REGION Network 42: Align Table Select Job
   // Decide which Step Sequence to start depending on the OMAC State and EM conditions
   // First Move Block is to Initialize the jobSelect Number
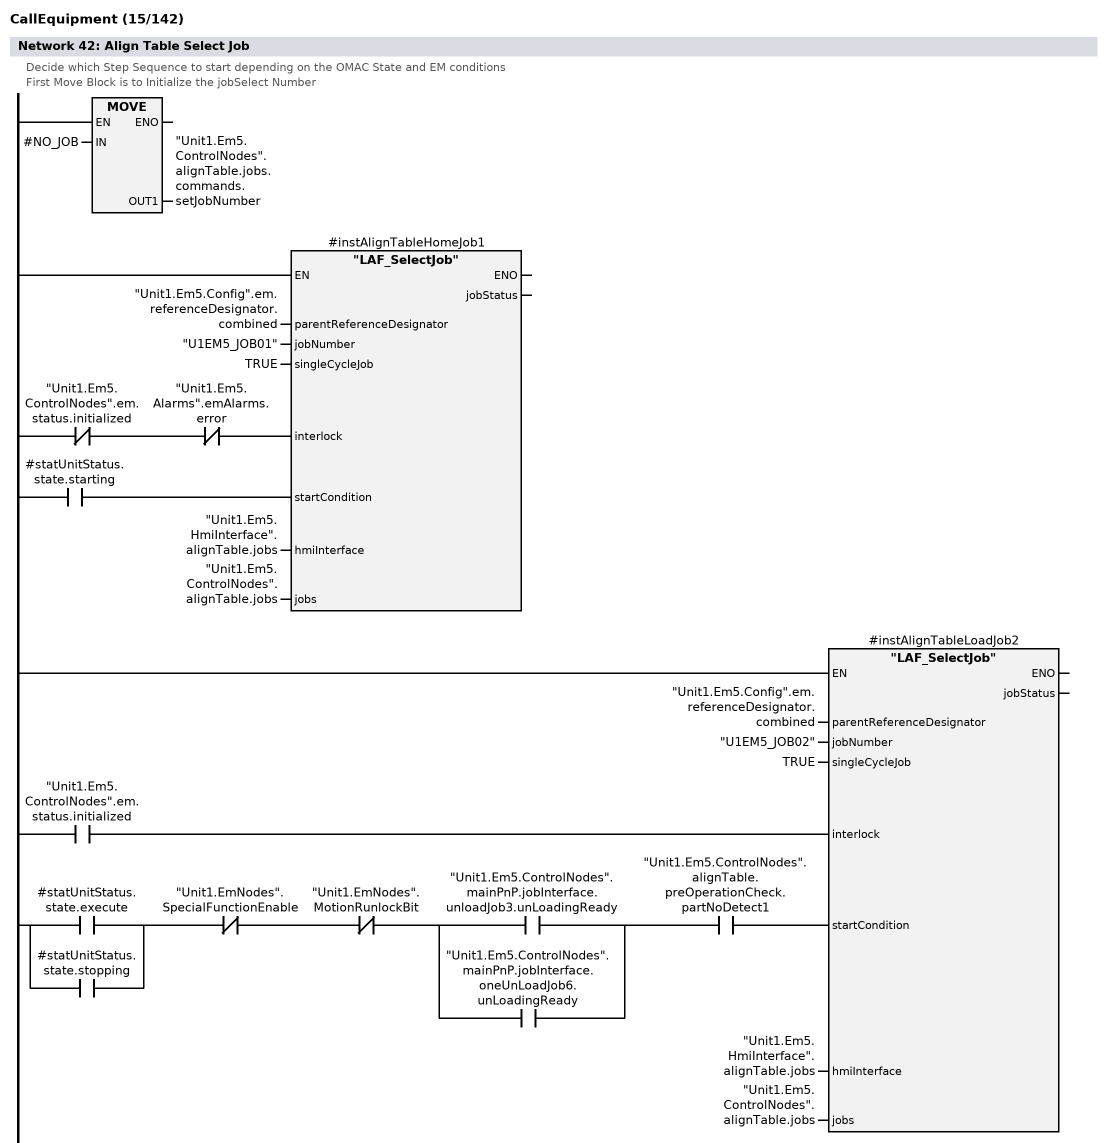
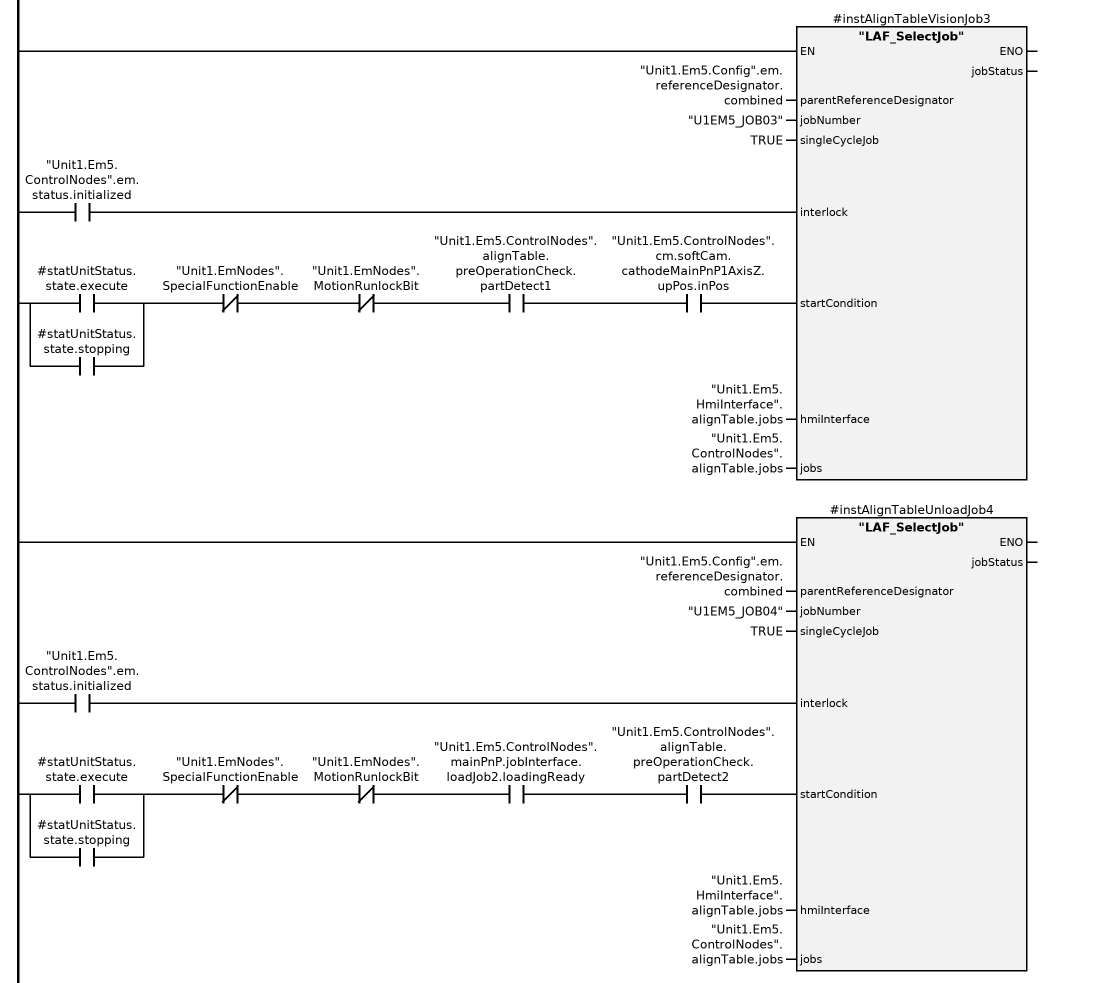
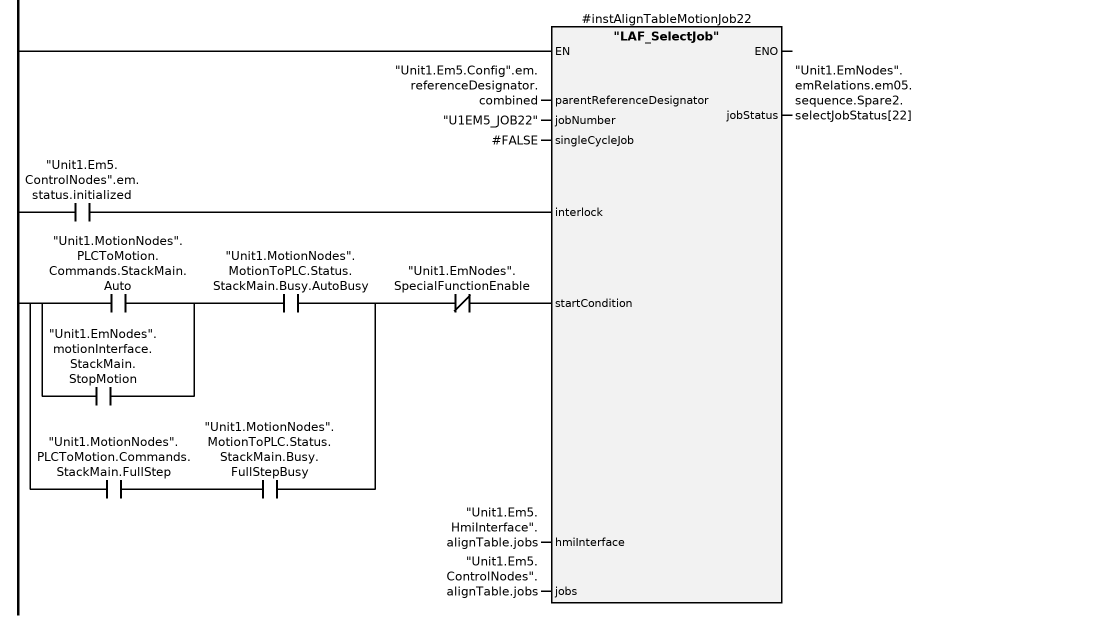
   RUNG wire#powerrail
      Move(in := #NO_JOB, out1 => "Unit1.Em5.ControlNodes".alignTable.jobs.commands.setJobNumber)
   END_RUNG
   RUNG wire#powerrail
      #instAlignTableHomeJob1(interlock := wire#w1, startCondition := wire#w2, parentReferenceDesignator := "Unit1.Em5.Config".em.referenceDesignator.combined, jobNumber := "U1EM5_JOB01", singleCycleJob := TRUE, hmiInterface := "Unit1.Em5.HmiInterface".alignTable.jobs, jobs := "Unit1.Em5.ControlNodes".alignTable.jobs, jobStatus =>)
   END_RUNG
   RUNG wire#powerrail
      I_Contact( "Unit1.Em5.ControlNodes".em.status.initialized )
      I_Contact( "Unit1.Em5.Alarms".emAlarms.error )
   END_RUNG wire#w1
   RUNG wire#powerrail
      Contact( #statUnitStatus.state.starting )
   END_RUNG wire#w2
   RUNG wire#powerrail
      #instAlignTableLoadJob2(interlock := wire#w3, startCondition := wire#w7, parentReferenceDesignator := "Unit1.Em5.Config".em.referenceDesignator.combined, jobNumber := "U1EM5_JOB02", singleCycleJob := TRUE, hmiInterface := "Unit1.Em5.HmiInterface".alignTable.jobs, jobs := "Unit1.Em5.ControlNodes".alignTable.jobs, jobStatus =>)
   END_RUNG
   RUNG wire#powerrail
      Contact( "Unit1.Em5.ControlNodes".em.status.initialized )
   END_RUNG wire#w3
   RUNG wire#powerrail
      Contact( #statUnitStatus.state.execute )
      wire#w4
      I_Contact( "Unit1.EmNodes".SpecialFunctionEnable )
      I_Contact( "Unit1.EmNodes".MotionRunlockBit )
      wire#w5
      Contact( "Unit1.Em5.ControlNodes".mainPnP.jobInterface.unloadJob3.unLoadingReady )
      wire#w6
      Contact( "Unit1.Em5.ControlNodes".alignTable.preOperationCheck.partNoDetect1 )
   END_RUNG wire#w7
   RUNG wire#powerrail
      Contact( #statUnitStatus.state.stopping )
   END_RUNG wire#w4
   RUNG wire#w5
      Contact( "Unit1.Em5.ControlNodes".mainPnP.jobInterface.oneUnLoadJob6.unLoadingReady )
   END_RUNG wire#w6
   RUNG wire#powerrail
      #instAlignTableVisionJob3(interlock := wire#w8, startCondition := wire#w10, parentReferenceDesignator := "Unit1.Em5.Config".em.referenceDesignator.combined, jobNumber := "U1EM5_JOB03", singleCycleJob := TRUE, hmiInterface := "Unit1.Em5.HmiInterface".alignTable.jobs, jobs := "Unit1.Em5.ControlNodes".alignTable.jobs, jobStatus =>)
   END_RUNG
   RUNG wire#powerrail
      Contact( "Unit1.Em5.ControlNodes".em.status.initialized )
   END_RUNG wire#w8
   RUNG wire#powerrail
      Contact( #statUnitStatus.state.execute )
      wire#w9
      I_Contact( "Unit1.EmNodes".SpecialFunctionEnable )
      I_Contact( "Unit1.EmNodes".MotionRunlockBit )
      Contact( "Unit1.Em5.ControlNodes".alignTable.preOperationCheck.partDetect1 )
      Contact( "Unit1.Em5.ControlNodes".cm.softCam.cathodeMainPnP1AxisZ.upPos.inPos )
   END_RUNG wire#w10
   RUNG wire#powerrail
      Contact( #statUnitStatus.state.stopping )
   END_RUNG wire#w9
   RUNG wire#powerrail
      #instAlignTableUnloadJob4(interlock := wire#w11, startCondition := wire#w13, parentReferenceDesignator := "Unit1.Em5.Config".em.referenceDesignator.combined, jobNumber := "U1EM5_JOB04", singleCycleJob := TRUE, hmiInterface := "Unit1.Em5.HmiInterface".alignTable.jobs, jobs := "Unit1.Em5.ControlNodes".alignTable.jobs, jobStatus =>)
   END_RUNG
   RUNG wire#powerrail
      Contact( "Unit1.Em5.ControlNodes".em.status.initialized )
   END_RUNG wire#w11
   RUNG wire#powerrail
      Contact( #statUnitStatus.state.execute )
      wire#w12
      I_Contact( "Unit1.EmNodes".SpecialFunctionEnable )
      I_Contact( "Unit1.EmNodes".MotionRunlockBit )
      Contact( "Unit1.Em5.ControlNodes".mainPnP.jobInterface.loadJob2.loadingReady )
      Contact( "Unit1.Em5.ControlNodes".alignTable.preOperationCheck.partDetect2 )
   END_RUNG wire#w13
   RUNG wire#powerrail
      Contact( #statUnitStatus.state.stopping )
   END_RUNG wire#w12
   RUNG wire#powerrail
      #instAlignTableMotionJob22(interlock := wire#w14, startCondition := wire#w17, parentReferenceDesignator := "Unit1.Em5.Config".em.referenceDesignator.combined, jobNumber := "U1EM5_JOB22", singleCycleJob := #FALSE, hmiInterface := "Unit1.Em5.HmiInterface".alignTable.jobs, jobs := "Unit1.Em5.ControlNodes".alignTable.jobs, jobStatus => "Unit1.EmNodes".emRelations.em05.sequence.Spare2.selectJobStatus[22])
   END_RUNG
   RUNG wire#powerrail
      Contact( "Unit1.Em5.ControlNodes".em.status.initialized )
   END_RUNG wire#w14
   RUNG wire#powerrail
      Contact( "Unit1.MotionNodes".PLCToMotion.Commands.StackMain.Auto )
      wire#w15
      Contact( "Unit1.MotionNodes".MotionToPLC.Status.StackMain.Busy.AutoBusy )
      wire#w16
      I_Contact( "Unit1.EmNodes".SpecialFunctionEnable )
   END_RUNG wire#w17
   RUNG wire#powerrail
      Contact( "Unit1.EmNodes".motionInterface.StackMain.StopMotion )
   END_RUNG wire#w15
   RUNG wire#powerrail
      Contact( "Unit1.MotionNodes".PLCToMotion.Commands.StackMain.FullStep )
      Contact( "Unit1.MotionNodes".MotionToPLC.Status.StackMain.Busy.FullStepBusy )
   END_RUNG wire#w16
   // the same network as SCL:
   "Unit1.Em5.ControlNodes".alignTable.jobs.commands.setJobNumber := #NO_JOB;
   #instAlignTableHomeJob1(parentReferenceDesignator := "Unit1.Em5.Config".em.referenceDesignator.combined,   // "LAF_SelectJob"
                           jobNumber := "U1EM5_JOB01",
                           singleCycleJob := TRUE,
                           interlock := NOT "Unit1.Em5.ControlNodes".em.status.initialized AND NOT "Unit1.Em5.Alarms".emAlarms.error,
                           startCondition := #statUnitStatus.state.starting,
                           hmiInterface := "Unit1.Em5.HmiInterface".alignTable.jobs,
                           jobs := "Unit1.Em5.ControlNodes".alignTable.jobs);
   #instAlignTableLoadJob2(parentReferenceDesignator := "Unit1.Em5.Config".em.referenceDesignator.combined,   // "LAF_SelectJob"
                           jobNumber := "U1EM5_JOB02",
                           singleCycleJob := TRUE,
                           interlock := "Unit1.Em5.ControlNodes".em.status.initialized,
                           startCondition := (#statUnitStatus.state.execute OR #statUnitStatus.state.stopping) AND NOT "Unit1.EmNodes".SpecialFunctionEnable AND NOT "Unit1.EmNodes".MotionRunlockBit AND ("Unit1.Em5.ControlNodes".mainPnP.jobInterface.unloadJob3.unLoadingReady OR "Unit1.Em5.ControlNodes".mainPnP.jobInterface.oneUnLoadJob6.unLoadingReady) AND "Unit1.Em5.ControlNodes".alignTable.preOperationCheck.partNoDetect1,
                           hmiInterface := "Unit1.Em5.HmiInterface".alignTable.jobs,
                           jobs := "Unit1.Em5.ControlNodes".alignTable.jobs);
   #instAlignTableVisionJob3(parentReferenceDesignator := "Unit1.Em5.Config".em.referenceDesignator.combined,   // "LAF_SelectJob"
                           jobNumber := "U1EM5_JOB03",
                           singleCycleJob := TRUE,
                           interlock := "Unit1.Em5.ControlNodes".em.status.initialized,
                           startCondition := (#statUnitStatus.state.execute OR #statUnitStatus.state.stopping) AND NOT "Unit1.EmNodes".SpecialFunctionEnable AND NOT "Unit1.EmNodes".MotionRunlockBit AND "Unit1.Em5.ControlNodes".alignTable.preOperationCheck.partDetect1 AND "Unit1.Em5.ControlNodes".cm.softCam.cathodeMainPnP1AxisZ.upPos.inPos,
                           hmiInterface := "Unit1.Em5.HmiInterface".alignTable.jobs,
                           jobs := "Unit1.Em5.ControlNodes".alignTable.jobs);
   #instAlignTableUnloadJob4(parentReferenceDesignator := "Unit1.Em5.Config".em.referenceDesignator.combined,   // "LAF_SelectJob"
                           jobNumber := "U1EM5_JOB04",
                           singleCycleJob := TRUE,
                           interlock := "Unit1.Em5.ControlNodes".em.status.initialized,
                           startCondition := (#statUnitStatus.state.execute OR #statUnitStatus.state.stopping) AND NOT "Unit1.EmNodes".SpecialFunctionEnable AND NOT "Unit1.EmNodes".MotionRunlockBit AND "Unit1.Em5.ControlNodes".mainPnP.jobInterface.loadJob2.loadingReady AND "Unit1.Em5.ControlNodes".alignTable.preOperationCheck.partDetect2,
                           hmiInterface := "Unit1.Em5.HmiInterface".alignTable.jobs,
                           jobs := "Unit1.Em5.ControlNodes".alignTable.jobs);
   #instAlignTableMotionJob22(parentReferenceDesignator := "Unit1.Em5.Config".em.referenceDesignator.combined,   // "LAF_SelectJob"
                           jobNumber := "U1EM5_JOB22",
                           singleCycleJob := #FALSE,
                           interlock := "Unit1.Em5.ControlNodes".em.status.initialized,
                           startCondition := ((("Unit1.MotionNodes".PLCToMotion.Commands.StackMain.Auto OR "Unit1.EmNodes".motionInterface.StackMain.StopMotion) AND "Unit1.MotionNodes".MotionToPLC.Status.StackMain.Busy.AutoBusy) OR ("Unit1.MotionNodes".PLCToMotion.Commands.StackMain.FullStep AND "Unit1.MotionNodes".MotionToPLC.Status.StackMain.Busy.FullStepBusy)) AND NOT "Unit1.EmNodes".SpecialFunctionEnable,
                           hmiInterface := "Unit1.Em5.HmiInterface".alignTable.jobs,
                           jobs := "Unit1.Em5.ControlNodes".alignTable.jobs,
                           jobStatus => "Unit1.EmNodes".emRelations.em05.sequence.Spare2.selectJobStatus[22]);
END_REGION

REGION Network 43: Align Table Job 1 Interface
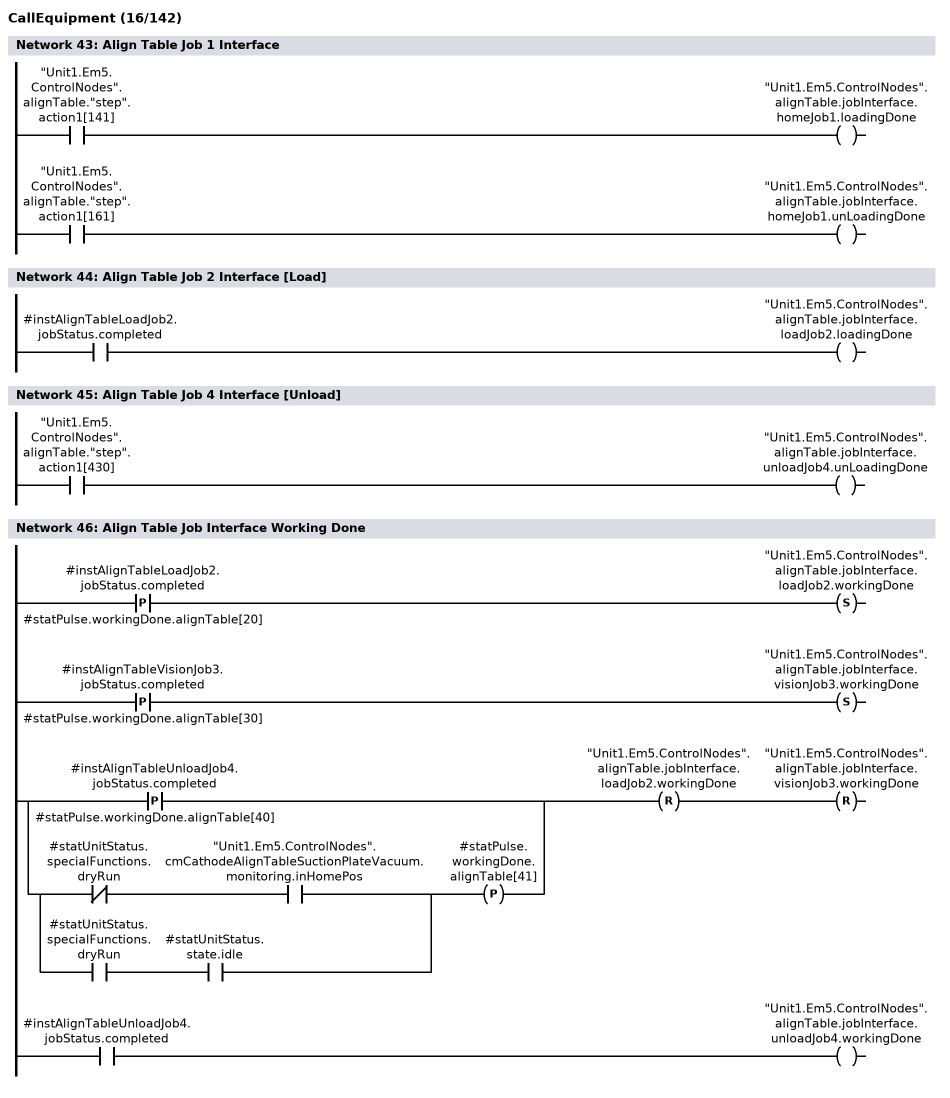
   RUNG wire#powerrail
      Contact( "Unit1.Em5.ControlNodes".alignTable."step".action1[141] )
      Coil( "Unit1.Em5.ControlNodes".alignTable.jobInterface.homeJob1.loadingDone )
   END_RUNG
   RUNG wire#powerrail
      Contact( "Unit1.Em5.ControlNodes".alignTable."step".action1[161] )
      Coil( "Unit1.Em5.ControlNodes".alignTable.jobInterface.homeJob1.unLoadingDone )
   END_RUNG
   // the same network as SCL:
   "Unit1.Em5.ControlNodes".alignTable.jobInterface.homeJob1.loadingDone := "Unit1.Em5.ControlNodes".alignTable."step".action1[141];
   "Unit1.Em5.ControlNodes".alignTable.jobInterface.homeJob1.unLoadingDone := "Unit1.Em5.ControlNodes".alignTable."step".action1[161];
END_REGION

REGION Network 44: Align Table Job 2 Interface [Load]
   RUNG wire#powerrail
      Contact( #instAlignTableLoadJob2.jobStatus.completed )
      Coil( "Unit1.Em5.ControlNodes".alignTable.jobInterface.loadJob2.loadingDone )
   END_RUNG
   // the same network as SCL:
   "Unit1.Em5.ControlNodes".alignTable.jobInterface.loadJob2.loadingDone := #instAlignTableLoadJob2.jobStatus.completed;
END_REGION

REGION Network 45: Align Table Job 4 Interface [Unload]
   RUNG wire#powerrail
      Contact( "Unit1.Em5.ControlNodes".alignTable."step".action1[430] )
      Coil( "Unit1.Em5.ControlNodes".alignTable.jobInterface.unloadJob4.unLoadingDone )
   END_RUNG
   // the same network as SCL:
   "Unit1.Em5.ControlNodes".alignTable.jobInterface.unloadJob4.unLoadingDone := "Unit1.Em5.ControlNodes".alignTable."step".action1[430];
END_REGION

REGION Network 46: Align Table Job Interface Working Done
   RUNG wire#powerrail
      P_Contact(operand := #instAlignTableLoadJob2.jobStatus.completed, bit := #statPulse.workingDone.alignTable[20])
      S_Coil( "Unit1.Em5.ControlNodes".alignTable.jobInterface.loadJob2.workingDone )
   END_RUNG
   RUNG wire#powerrail
      P_Contact(operand := #instAlignTableVisionJob3.jobStatus.completed, bit := #statPulse.workingDone.alignTable[30])
      S_Coil( "Unit1.Em5.ControlNodes".alignTable.jobInterface.visionJob3.workingDone )
   END_RUNG
   RUNG wire#powerrail
      P_Contact(operand := #instAlignTableUnloadJob4.jobStatus.completed, bit := #statPulse.workingDone.alignTable[40])
      wire#w1
      R_Coil( "Unit1.Em5.ControlNodes".alignTable.jobInterface.loadJob2.workingDone )
      R_Coil( "Unit1.Em5.ControlNodes".alignTable.jobInterface.visionJob3.workingDone )
   END_RUNG
   RUNG wire#powerrail
      I_Contact( #statUnitStatus.specialFunctions.dryRun )
      Contact( "Unit1.Em5.ControlNodes".cmCathodeAlignTableSuctionPlateVacuum.monitoring.inHomePos )
      wire#w2
      P_Trig( #statPulse.workingDone.alignTable[41] )
   END_RUNG wire#w1
   RUNG wire#powerrail
      Contact( #statUnitStatus.specialFunctions.dryRun )
      Contact( #statUnitStatus.state.idle )
   END_RUNG wire#w2
   RUNG wire#powerrail
      Contact( #instAlignTableUnloadJob4.jobStatus.completed )
      Coil( "Unit1.Em5.ControlNodes".alignTable.jobInterface.unloadJob4.workingDone )
   END_RUNG
   // the same network as SCL:
   #_w1 := #instAlignTableLoadJob2.jobStatus.completed AND NOT #statPulse.workingDone.alignTable[20];   // rising edge of #instAlignTableLoadJob2.jobStatus.completed
   #statPulse.workingDone.alignTable[20] := #instAlignTableLoadJob2.jobStatus.completed;
   IF #_w1 THEN "Unit1.Em5.ControlNodes".alignTable.jobInterface.loadJob2.workingDone := TRUE; END_IF;
   #_w2 := #instAlignTableVisionJob3.jobStatus.completed AND NOT #statPulse.workingDone.alignTable[30];   // rising edge of #instAlignTableVisionJob3.jobStatus.completed
   #statPulse.workingDone.alignTable[30] := #instAlignTableVisionJob3.jobStatus.completed;
   IF #_w2 THEN "Unit1.Em5.ControlNodes".alignTable.jobInterface.visionJob3.workingDone := TRUE; END_IF;
   #_w3 := #instAlignTableUnloadJob4.jobStatus.completed AND NOT #statPulse.workingDone.alignTable[40];   // rising edge of #instAlignTableUnloadJob4.jobStatus.completed
   #statPulse.workingDone.alignTable[40] := #instAlignTableUnloadJob4.jobStatus.completed;
   #_w4 := (NOT #statUnitStatus.specialFunctions.dryRun AND "Unit1.Em5.ControlNodes".cmCathodeAlignTableSuctionPlateVacuum.monitoring.inHomePos) OR (#statUnitStatus.specialFunctions.dryRun AND #statUnitStatus.state.idle);
   #_w5 := #_w4 AND NOT #statPulse.workingDone.alignTable[41];   // rising edge
   #statPulse.workingDone.alignTable[41] := #_w4;
   IF #_w3 OR #_w5 THEN
       "Unit1.Em5.ControlNodes".alignTable.jobInterface.loadJob2.workingDone := FALSE;
       "Unit1.Em5.ControlNodes".alignTable.jobInterface.visionJob3.workingDone := FALSE;
   END_IF;
   "Unit1.Em5.ControlNodes".alignTable.jobInterface.unloadJob4.workingDone := #instAlignTableUnloadJob4.jobStatus.completed;
END_REGION

REGION Network 47: Align Table Previous Operation Check
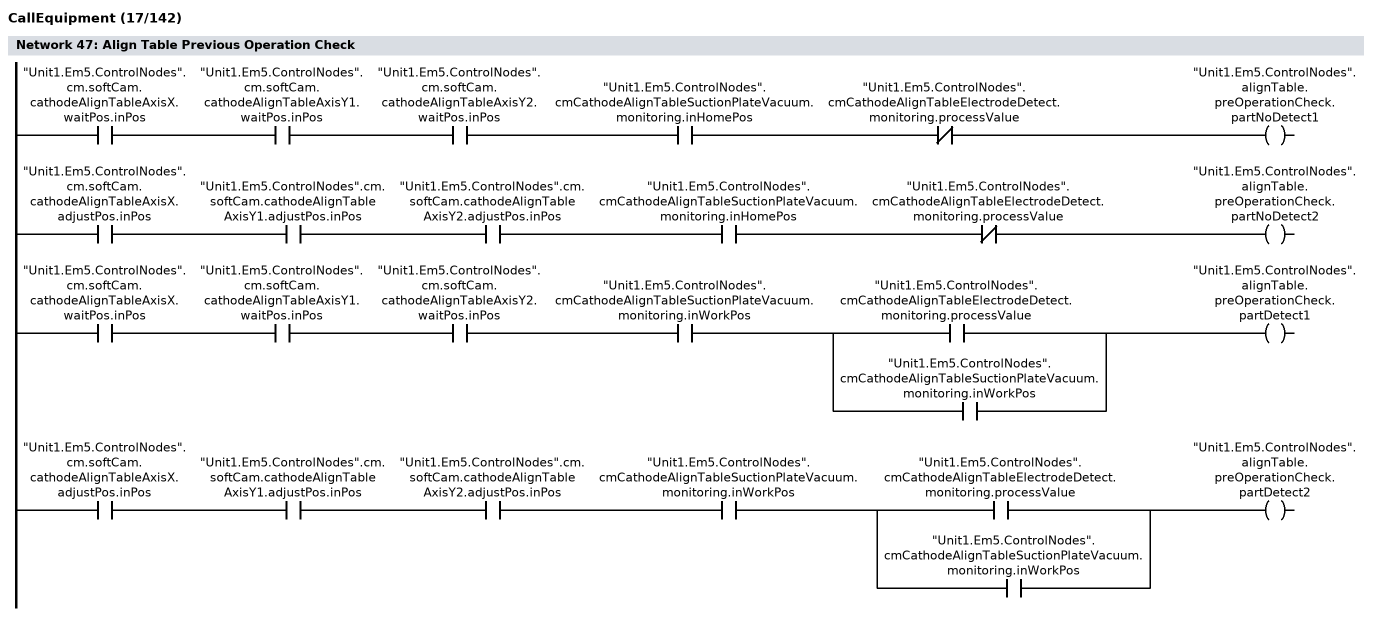
   RUNG wire#powerrail
      Contact( "Unit1.Em5.ControlNodes".cm.softCam.cathodeAlignTableAxisX.waitPos.inPos )
      Contact( "Unit1.Em5.ControlNodes".cm.softCam.cathodeAlignTableAxisY1.waitPos.inPos )
      Contact( "Unit1.Em5.ControlNodes".cm.softCam.cathodeAlignTableAxisY2.waitPos.inPos )
      Contact( "Unit1.Em5.ControlNodes".cmCathodeAlignTableSuctionPlateVacuum.monitoring.inHomePos )
      I_Contact( "Unit1.Em5.ControlNodes".cmCathodeAlignTableElectrodeDetect.monitoring.processValue )
      Coil( "Unit1.Em5.ControlNodes".alignTable.preOperationCheck.partNoDetect1 )
   END_RUNG
   RUNG wire#powerrail
      Contact( "Unit1.Em5.ControlNodes".cm.softCam.cathodeAlignTableAxisX.adjustPos.inPos )
      Contact( "Unit1.Em5.ControlNodes".cm.softCam.cathodeAlignTableAxisY1.adjustPos.inPos )
      Contact( "Unit1.Em5.ControlNodes".cm.softCam.cathodeAlignTableAxisY2.adjustPos.inPos )
      Contact( "Unit1.Em5.ControlNodes".cmCathodeAlignTableSuctionPlateVacuum.monitoring.inHomePos )
      I_Contact( "Unit1.Em5.ControlNodes".cmCathodeAlignTableElectrodeDetect.monitoring.processValue )
      Coil( "Unit1.Em5.ControlNodes".alignTable.preOperationCheck.partNoDetect2 )
   END_RUNG
   RUNG wire#powerrail
      Contact( "Unit1.Em5.ControlNodes".cm.softCam.cathodeAlignTableAxisX.waitPos.inPos )
      Contact( "Unit1.Em5.ControlNodes".cm.softCam.cathodeAlignTableAxisY1.waitPos.inPos )
      Contact( "Unit1.Em5.ControlNodes".cm.softCam.cathodeAlignTableAxisY2.waitPos.inPos )
      Contact( "Unit1.Em5.ControlNodes".cmCathodeAlignTableSuctionPlateVacuum.monitoring.inWorkPos )
      wire#w1
      Contact( "Unit1.Em5.ControlNodes".cmCathodeAlignTableElectrodeDetect.monitoring.processValue )
      wire#w2
      Coil( "Unit1.Em5.ControlNodes".alignTable.preOperationCheck.partDetect1 )
   END_RUNG
   RUNG wire#w1
      Contact( "Unit1.Em5.ControlNodes".cmCathodeAlignTableSuctionPlateVacuum.monitoring.inWorkPos )
   END_RUNG wire#w2
   RUNG wire#powerrail
      Contact( "Unit1.Em5.ControlNodes".cm.softCam.cathodeAlignTableAxisX.adjustPos.inPos )
      Contact( "Unit1.Em5.ControlNodes".cm.softCam.cathodeAlignTableAxisY1.adjustPos.inPos )
      Contact( "Unit1.Em5.ControlNodes".cm.softCam.cathodeAlignTableAxisY2.adjustPos.inPos )
      Contact( "Unit1.Em5.ControlNodes".cmCathodeAlignTableSuctionPlateVacuum.monitoring.inWorkPos )
      wire#w3
      Contact( "Unit1.Em5.ControlNodes".cmCathodeAlignTableElectrodeDetect.monitoring.processValue )
      wire#w4
      Coil( "Unit1.Em5.ControlNodes".alignTable.preOperationCheck.partDetect2 )
   END_RUNG
   RUNG wire#w3
      Contact( "Unit1.Em5.ControlNodes".cmCathodeAlignTableSuctionPlateVacuum.monitoring.inWorkPos )
   END_RUNG wire#w4
   // the same network as SCL:
   "Unit1.Em5.ControlNodes".alignTable.preOperationCheck.partNoDetect1 := "Unit1.Em5.ControlNodes".cm.softCam.cathodeAlignTableAxisX.waitPos.inPos AND "Unit1.Em5.ControlNodes".cm.softCam.cathodeAlignTableAxisY1.waitPos.inPos AND "Unit1.Em5.ControlNodes".cm.softCam.cathodeAlignTableAxisY2.waitPos.inPos AND "Unit1.Em5.ControlNodes".cmCathodeAlignTableSuctionPlateVacuum.monitoring.inHomePos AND NOT "Unit1.Em5.ControlNodes".cmCathodeAlignTableElectrodeDetect.monitoring.processValue;
   "Unit1.Em5.ControlNodes".alignTable.preOperationCheck.partNoDetect2 := "Unit1.Em5.ControlNodes".cm.softCam.cathodeAlignTableAxisX.adjustPos.inPos AND "Unit1.Em5.ControlNodes".cm.softCam.cathodeAlignTableAxisY1.adjustPos.inPos AND "Unit1.Em5.ControlNodes".cm.softCam.cathodeAlignTableAxisY2.adjustPos.inPos AND "Unit1.Em5.ControlNodes".cmCathodeAlignTableSuctionPlateVacuum.monitoring.inHomePos AND NOT "Unit1.Em5.ControlNodes".cmCathodeAlignTableElectrodeDetect.monitoring.processValue;
   "Unit1.Em5.ControlNodes".alignTable.preOperationCheck.partDetect1 := "Unit1.Em5.ControlNodes".cm.softCam.cathodeAlignTableAxisX.waitPos.inPos AND "Unit1.Em5.ControlNodes".cm.softCam.cathodeAlignTableAxisY1.waitPos.inPos AND "Unit1.Em5.ControlNodes".cm.softCam.cathodeAlignTableAxisY2.waitPos.inPos AND "Unit1.Em5.ControlNodes".cmCathodeAlignTableSuctionPlateVacuum.monitoring.inWorkPos AND ("Unit1.Em5.ControlNodes".cmCathodeAlignTableElectrodeDetect.monitoring.processValue OR "Unit1.Em5.ControlNodes".cmCathodeAlignTableSuctionPlateVacuum.monitoring.inWorkPos);
   "Unit1.Em5.ControlNodes".alignTable.preOperationCheck.partDetect2 := "Unit1.Em5.ControlNodes".cm.softCam.cathodeAlignTableAxisX.adjustPos.inPos AND "Unit1.Em5.ControlNodes".cm.softCam.cathodeAlignTableAxisY1.adjustPos.inPos AND "Unit1.Em5.ControlNodes".cm.softCam.cathodeAlignTableAxisY2.adjustPos.inPos AND "Unit1.Em5.ControlNodes".cmCathodeAlignTableSuctionPlateVacuum.monitoring.inWorkPos AND ("Unit1.Em5.ControlNodes".cmCathodeAlignTableElectrodeDetect.monitoring.processValue OR "Unit1.Em5.ControlNodes".cmCathodeAlignTableSuctionPlateVacuum.monitoring.inWorkPos);
END_REGION

REGION Network 49: NG P&P Select Job
   // Decide which Step Sequence to start depending on the OMAC State and EM conditions
   // First Move Block is to Initialize the jobSelect Number
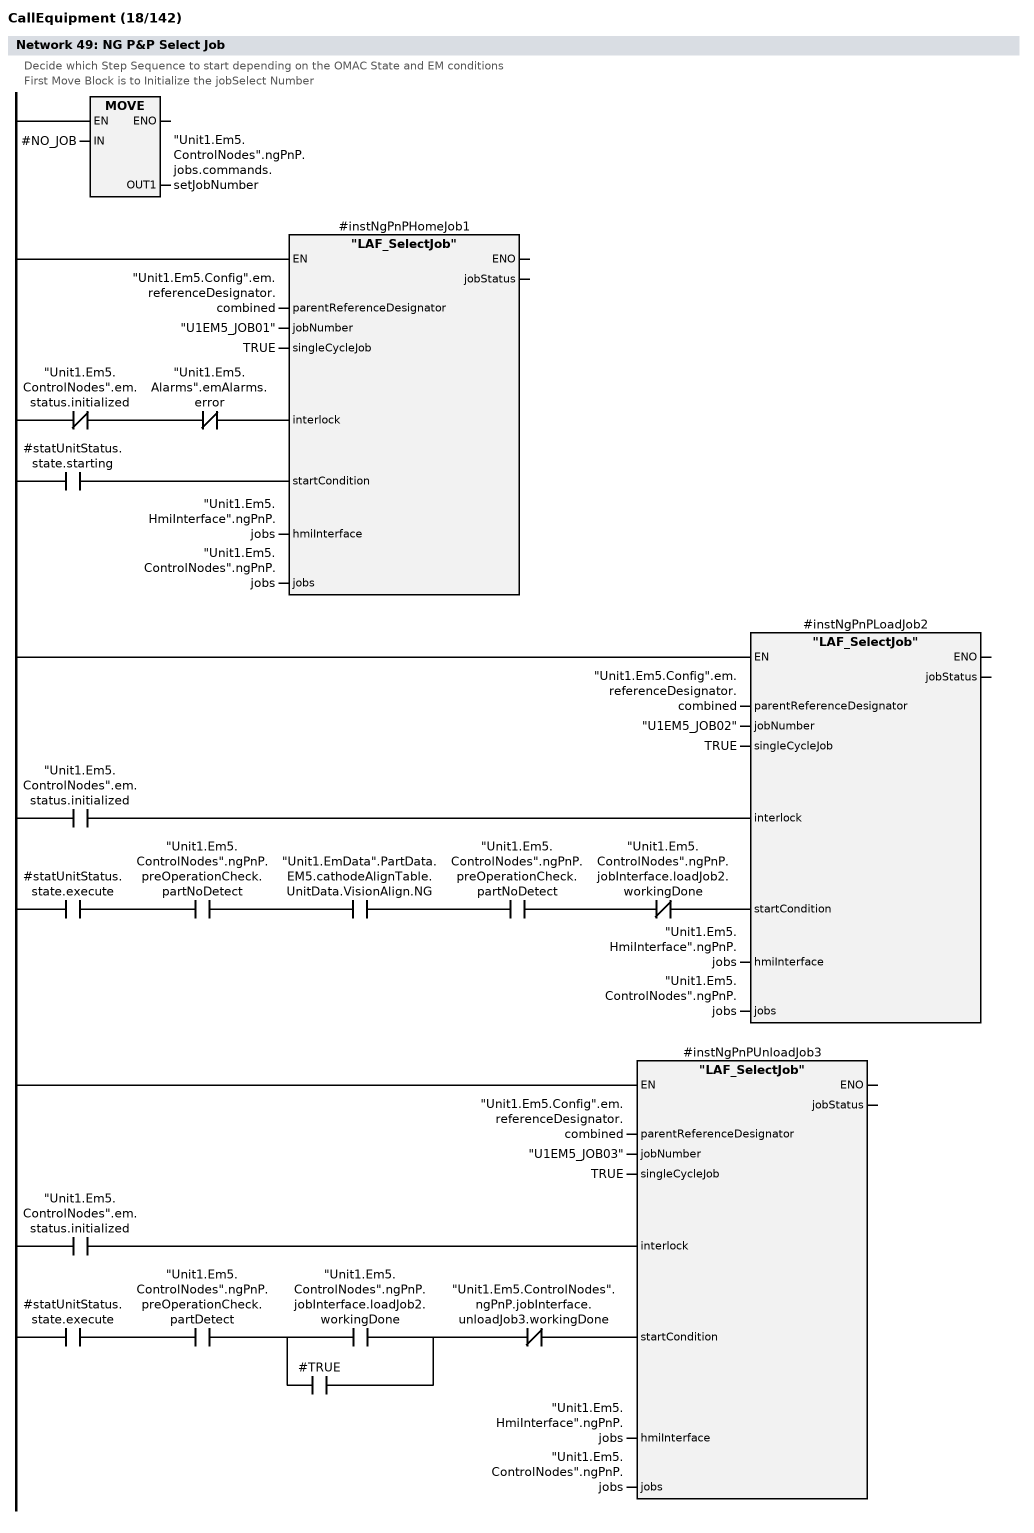
   RUNG wire#powerrail
      Move(in := #NO_JOB, out1 => "Unit1.Em5.ControlNodes".ngPnP.jobs.commands.setJobNumber)
   END_RUNG
   RUNG wire#powerrail
      #instNgPnPHomeJob1(interlock := wire#w1, startCondition := wire#w2, parentReferenceDesignator := "Unit1.Em5.Config".em.referenceDesignator.combined, jobNumber := "U1EM5_JOB01", singleCycleJob := TRUE, hmiInterface := "Unit1.Em5.HmiInterface".ngPnP.jobs, jobs := "Unit1.Em5.ControlNodes".ngPnP.jobs, jobStatus =>)
   END_RUNG
   RUNG wire#powerrail
      I_Contact( "Unit1.Em5.ControlNodes".em.status.initialized )
      I_Contact( "Unit1.Em5.Alarms".emAlarms.error )
   END_RUNG wire#w1
   RUNG wire#powerrail
      Contact( #statUnitStatus.state.starting )
   END_RUNG wire#w2
   RUNG wire#powerrail
      #instNgPnPLoadJob2(interlock := wire#w3, startCondition := wire#w4, parentReferenceDesignator := "Unit1.Em5.Config".em.referenceDesignator.combined, jobNumber := "U1EM5_JOB02", singleCycleJob := TRUE, hmiInterface := "Unit1.Em5.HmiInterface".ngPnP.jobs, jobs := "Unit1.Em5.ControlNodes".ngPnP.jobs, jobStatus =>)
   END_RUNG
   RUNG wire#powerrail
      Contact( "Unit1.Em5.ControlNodes".em.status.initialized )
   END_RUNG wire#w3
   RUNG wire#powerrail
      Contact( #statUnitStatus.state.execute )
      Contact( "Unit1.Em5.ControlNodes".ngPnP.preOperationCheck.partNoDetect )
      Contact( "Unit1.EmData".PartData.EM5.cathodeAlignTable.UnitData.VisionAlign.NG )
      Contact( "Unit1.Em5.ControlNodes".ngPnP.preOperationCheck.partNoDetect )
      I_Contact( "Unit1.Em5.ControlNodes".ngPnP.jobInterface.loadJob2.workingDone )
   END_RUNG wire#w4
   RUNG wire#powerrail
      #instNgPnPUnloadJob3(interlock := wire#w5, startCondition := wire#w8, parentReferenceDesignator := "Unit1.Em5.Config".em.referenceDesignator.combined, jobNumber := "U1EM5_JOB03", singleCycleJob := TRUE, hmiInterface := "Unit1.Em5.HmiInterface".ngPnP.jobs, jobs := "Unit1.Em5.ControlNodes".ngPnP.jobs, jobStatus =>)
   END_RUNG
   RUNG wire#powerrail
      Contact( "Unit1.Em5.ControlNodes".em.status.initialized )
   END_RUNG wire#w5
   RUNG wire#powerrail
      Contact( #statUnitStatus.state.execute )
      Contact( "Unit1.Em5.ControlNodes".ngPnP.preOperationCheck.partDetect )
      wire#w6
      Contact( "Unit1.Em5.ControlNodes".ngPnP.jobInterface.loadJob2.workingDone )
      wire#w7
      I_Contact( "Unit1.Em5.ControlNodes".ngPnP.jobInterface.unloadJob3.workingDone )
   END_RUNG wire#w8
   RUNG wire#w6
      Contact( #TRUE )
   END_RUNG wire#w7
   // the same network as SCL:
   "Unit1.Em5.ControlNodes".ngPnP.jobs.commands.setJobNumber := #NO_JOB;
   #instNgPnPHomeJob1(parentReferenceDesignator := "Unit1.Em5.Config".em.referenceDesignator.combined,   // "LAF_SelectJob"
                      jobNumber := "U1EM5_JOB01",
                      singleCycleJob := TRUE,
                      interlock := NOT "Unit1.Em5.ControlNodes".em.status.initialized AND NOT "Unit1.Em5.Alarms".emAlarms.error,
                      startCondition := #statUnitStatus.state.starting,
                      hmiInterface := "Unit1.Em5.HmiInterface".ngPnP.jobs,
                      jobs := "Unit1.Em5.ControlNodes".ngPnP.jobs);
   #instNgPnPLoadJob2(parentReferenceDesignator := "Unit1.Em5.Config".em.referenceDesignator.combined,   // "LAF_SelectJob"
                      jobNumber := "U1EM5_JOB02",
                      singleCycleJob := TRUE,
                      interlock := "Unit1.Em5.ControlNodes".em.status.initialized,
                      startCondition := #statUnitStatus.state.execute AND "Unit1.Em5.ControlNodes".ngPnP.preOperationCheck.partNoDetect AND "Unit1.EmData".PartData.EM5.cathodeAlignTable.UnitData.VisionAlign.NG AND "Unit1.Em5.ControlNodes".ngPnP.preOperationCheck.partNoDetect AND NOT "Unit1.Em5.ControlNodes".ngPnP.jobInterface.loadJob2.workingDone,
                      hmiInterface := "Unit1.Em5.HmiInterface".ngPnP.jobs,
                      jobs := "Unit1.Em5.ControlNodes".ngPnP.jobs);
   #instNgPnPUnloadJob3(parentReferenceDesignator := "Unit1.Em5.Config".em.referenceDesignator.combined,   // "LAF_SelectJob"
                        jobNumber := "U1EM5_JOB03",
                        singleCycleJob := TRUE,
                        interlock := "Unit1.Em5.ControlNodes".em.status.initialized,
                        startCondition := #statUnitStatus.state.execute AND "Unit1.Em5.ControlNodes".ngPnP.preOperationCheck.partDetect AND ("Unit1.Em5.ControlNodes".ngPnP.jobInterface.loadJob2.workingDone OR #TRUE) AND NOT "Unit1.Em5.ControlNodes".ngPnP.jobInterface.unloadJob3.workingDone,
                        hmiInterface := "Unit1.Em5.HmiInterface".ngPnP.jobs,
                        jobs := "Unit1.Em5.ControlNodes".ngPnP.jobs);
END_REGION

REGION Network 50: NG P&P Job 1 Interface
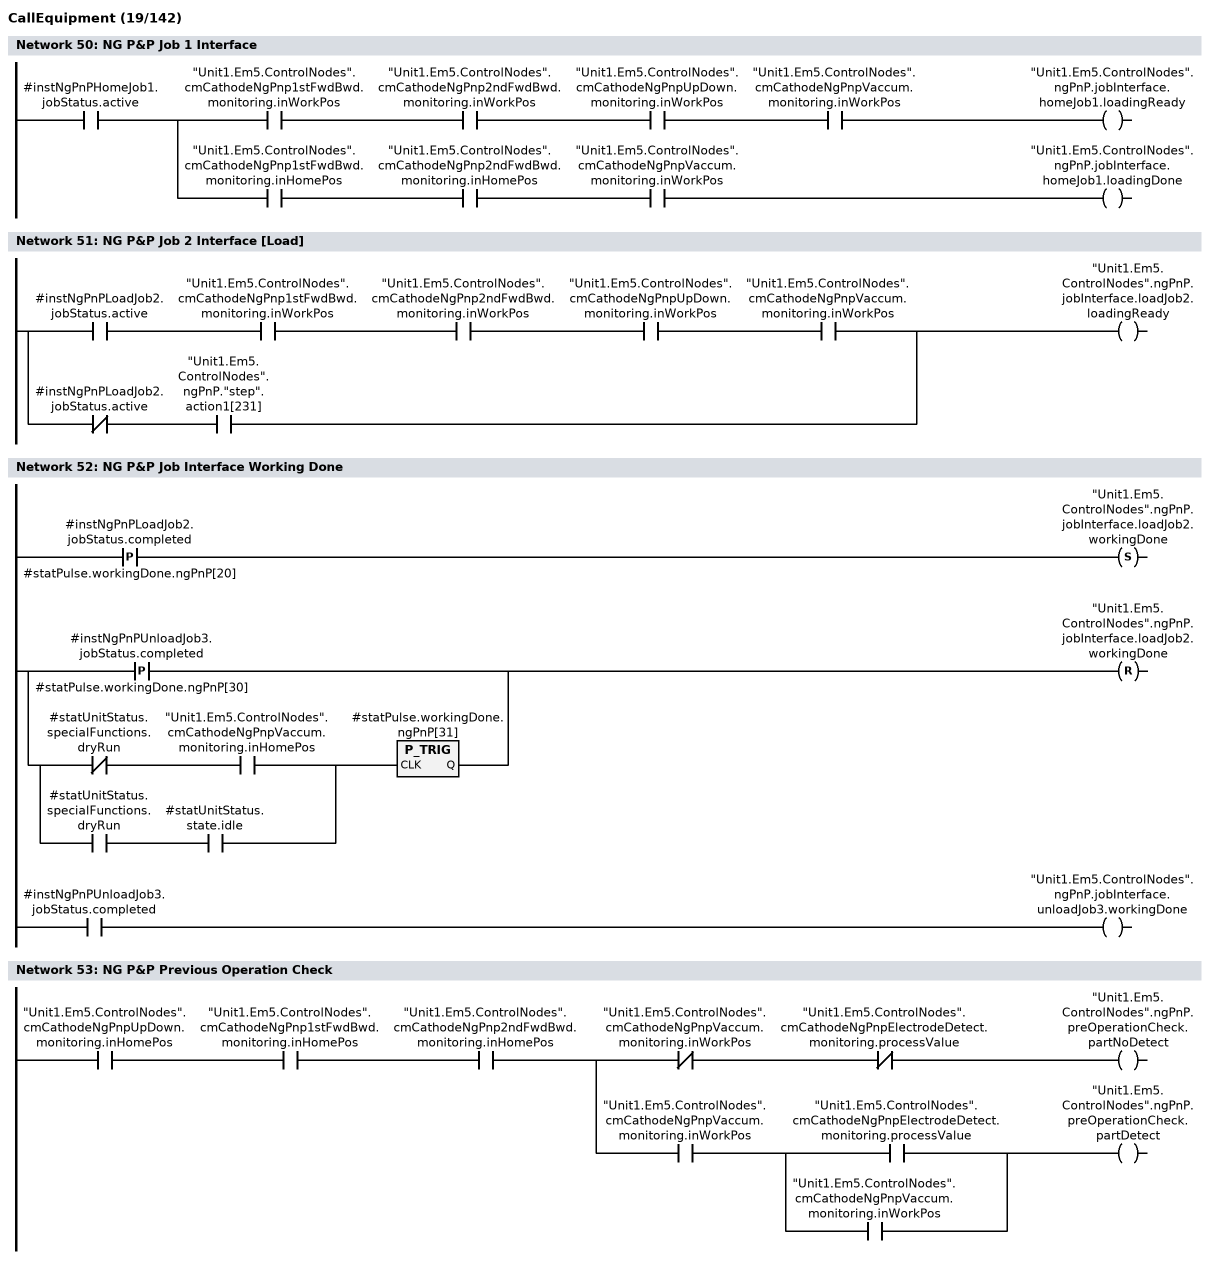
   RUNG wire#powerrail
      Contact( #instNgPnPHomeJob1.jobStatus.active )
      wire#w1
      Contact( "Unit1.Em5.ControlNodes".cmCathodeNgPnp1stFwdBwd.monitoring.inWorkPos )
      Contact( "Unit1.Em5.ControlNodes".cmCathodeNgPnp2ndFwdBwd.monitoring.inWorkPos )
      Contact( "Unit1.Em5.ControlNodes".cmCathodeNgPnpUpDown.monitoring.inWorkPos )
      Contact( "Unit1.Em5.ControlNodes".cmCathodeNgPnpVaccum.monitoring.inWorkPos )
      Coil( "Unit1.Em5.ControlNodes".ngPnP.jobInterface.homeJob1.loadingReady )
   END_RUNG
   RUNG wire#w1
      Contact( "Unit1.Em5.ControlNodes".cmCathodeNgPnp1stFwdBwd.monitoring.inHomePos )
      Contact( "Unit1.Em5.ControlNodes".cmCathodeNgPnp2ndFwdBwd.monitoring.inHomePos )
      Contact( "Unit1.Em5.ControlNodes".cmCathodeNgPnpVaccum.monitoring.inWorkPos )
      Coil( "Unit1.Em5.ControlNodes".ngPnP.jobInterface.homeJob1.loadingDone )
   END_RUNG
   // the same network as SCL:
   "Unit1.Em5.ControlNodes".ngPnP.jobInterface.homeJob1.loadingReady := #instNgPnPHomeJob1.jobStatus.active AND "Unit1.Em5.ControlNodes".cmCathodeNgPnp1stFwdBwd.monitoring.inWorkPos AND "Unit1.Em5.ControlNodes".cmCathodeNgPnp2ndFwdBwd.monitoring.inWorkPos AND "Unit1.Em5.ControlNodes".cmCathodeNgPnpUpDown.monitoring.inWorkPos AND "Unit1.Em5.ControlNodes".cmCathodeNgPnpVaccum.monitoring.inWorkPos;
   "Unit1.Em5.ControlNodes".ngPnP.jobInterface.homeJob1.loadingDone := #instNgPnPHomeJob1.jobStatus.active AND "Unit1.Em5.ControlNodes".cmCathodeNgPnp1stFwdBwd.monitoring.inHomePos AND "Unit1.Em5.ControlNodes".cmCathodeNgPnp2ndFwdBwd.monitoring.inHomePos AND "Unit1.Em5.ControlNodes".cmCathodeNgPnpVaccum.monitoring.inWorkPos;
END_REGION

REGION Network 51: NG P&P Job 2 Interface [Load]
   RUNG wire#powerrail
      Contact( #instNgPnPLoadJob2.jobStatus.active )
      Contact( "Unit1.Em5.ControlNodes".cmCathodeNgPnp1stFwdBwd.monitoring.inWorkPos )
      Contact( "Unit1.Em5.ControlNodes".cmCathodeNgPnp2ndFwdBwd.monitoring.inWorkPos )
      Contact( "Unit1.Em5.ControlNodes".cmCathodeNgPnpUpDown.monitoring.inWorkPos )
      Contact( "Unit1.Em5.ControlNodes".cmCathodeNgPnpVaccum.monitoring.inWorkPos )
      wire#w1
      Coil( "Unit1.Em5.ControlNodes".ngPnP.jobInterface.loadJob2.loadingReady )
   END_RUNG
   RUNG wire#powerrail
      I_Contact( #instNgPnPLoadJob2.jobStatus.active )
      Contact( "Unit1.Em5.ControlNodes".ngPnP."step".action1[231] )
   END_RUNG wire#w1
   // the same network as SCL:
   "Unit1.Em5.ControlNodes".ngPnP.jobInterface.loadJob2.loadingReady := (#instNgPnPLoadJob2.jobStatus.active AND "Unit1.Em5.ControlNodes".cmCathodeNgPnp1stFwdBwd.monitoring.inWorkPos AND "Unit1.Em5.ControlNodes".cmCathodeNgPnp2ndFwdBwd.monitoring.inWorkPos AND "Unit1.Em5.ControlNodes".cmCathodeNgPnpUpDown.monitoring.inWorkPos AND "Unit1.Em5.ControlNodes".cmCathodeNgPnpVaccum.monitoring.inWorkPos) OR (NOT #instNgPnPLoadJob2.jobStatus.active AND "Unit1.Em5.ControlNodes".ngPnP."step".action1[231]);
END_REGION

REGION Network 52: NG P&P Job Interface Working Done
   RUNG wire#powerrail
      P_Contact(operand := #instNgPnPLoadJob2.jobStatus.completed, bit := #statPulse.workingDone.ngPnP[20])
      S_Coil( "Unit1.Em5.ControlNodes".ngPnP.jobInterface.loadJob2.workingDone )
   END_RUNG
   RUNG wire#powerrail
      P_Contact(operand := #instNgPnPUnloadJob3.jobStatus.completed, bit := #statPulse.workingDone.ngPnP[30])
      wire#w1
      R_Coil( "Unit1.Em5.ControlNodes".ngPnP.jobInterface.loadJob2.workingDone )
   END_RUNG
   RUNG wire#powerrail
      I_Contact( #statUnitStatus.specialFunctions.dryRun )
      Contact( "Unit1.Em5.ControlNodes".cmCathodeNgPnpVaccum.monitoring.inHomePos )
      wire#w2
      P_Trig( #statPulse.workingDone.ngPnP[31] )
   END_RUNG wire#w1
   RUNG wire#powerrail
      Contact( #statUnitStatus.specialFunctions.dryRun )
      Contact( #statUnitStatus.state.idle )
   END_RUNG wire#w2
   RUNG wire#powerrail
      Contact( #instNgPnPUnloadJob3.jobStatus.completed )
      Coil( "Unit1.Em5.ControlNodes".ngPnP.jobInterface.unloadJob3.workingDone )
   END_RUNG
   // the same network as SCL:
   #_w1 := #instNgPnPLoadJob2.jobStatus.completed AND NOT #statPulse.workingDone.ngPnP[20];   // rising edge of #instNgPnPLoadJob2.jobStatus.completed
   #statPulse.workingDone.ngPnP[20] := #instNgPnPLoadJob2.jobStatus.completed;
   IF #_w1 THEN "Unit1.Em5.ControlNodes".ngPnP.jobInterface.loadJob2.workingDone := TRUE; END_IF;
   #_w2 := #instNgPnPUnloadJob3.jobStatus.completed AND NOT #statPulse.workingDone.ngPnP[30];   // rising edge of #instNgPnPUnloadJob3.jobStatus.completed
   #statPulse.workingDone.ngPnP[30] := #instNgPnPUnloadJob3.jobStatus.completed;
   #_w3 := (NOT #statUnitStatus.specialFunctions.dryRun AND "Unit1.Em5.ControlNodes".cmCathodeNgPnpVaccum.monitoring.inHomePos) OR (#statUnitStatus.specialFunctions.dryRun AND #statUnitStatus.state.idle);
   #_w4 := #_w3 AND NOT #statPulse.workingDone.ngPnP[31];   // rising edge
   #statPulse.workingDone.ngPnP[31] := #_w3;
   IF #_w2 OR #_w4 THEN "Unit1.Em5.ControlNodes".ngPnP.jobInterface.loadJob2.workingDone := FALSE; END_IF;
   "Unit1.Em5.ControlNodes".ngPnP.jobInterface.unloadJob3.workingDone := #instNgPnPUnloadJob3.jobStatus.completed;
END_REGION

REGION Network 53: NG P&P Previous Operation Check
   RUNG wire#powerrail
      Contact( "Unit1.Em5.ControlNodes".cmCathodeNgPnpUpDown.monitoring.inHomePos )
      Contact( "Unit1.Em5.ControlNodes".cmCathodeNgPnp1stFwdBwd.monitoring.inHomePos )
      Contact( "Unit1.Em5.ControlNodes".cmCathodeNgPnp2ndFwdBwd.monitoring.inHomePos )
      wire#w1
      I_Contact( "Unit1.Em5.ControlNodes".cmCathodeNgPnpVaccum.monitoring.inWorkPos )
      I_Contact( "Unit1.Em5.ControlNodes".cmCathodeNgPnpElectrodeDetect.monitoring.processValue )
      Coil( "Unit1.Em5.ControlNodes".ngPnP.preOperationCheck.partNoDetect )
   END_RUNG
   RUNG wire#w1
      Contact( "Unit1.Em5.ControlNodes".cmCathodeNgPnpVaccum.monitoring.inWorkPos )
      wire#w2
      Contact( "Unit1.Em5.ControlNodes".cmCathodeNgPnpElectrodeDetect.monitoring.processValue )
      wire#w3
      Coil( "Unit1.Em5.ControlNodes".ngPnP.preOperationCheck.partDetect )
   END_RUNG
   RUNG wire#w2
      Contact( "Unit1.Em5.ControlNodes".cmCathodeNgPnpVaccum.monitoring.inWorkPos )
   END_RUNG wire#w3
   // the same network as SCL:
   #_w1 := "Unit1.Em5.ControlNodes".cmCathodeNgPnpUpDown.monitoring.inHomePos AND "Unit1.Em5.ControlNodes".cmCathodeNgPnp1stFwdBwd.monitoring.inHomePos AND "Unit1.Em5.ControlNodes".cmCathodeNgPnp2ndFwdBwd.monitoring.inHomePos;
   "Unit1.Em5.ControlNodes".ngPnP.preOperationCheck.partNoDetect := #_w1 AND NOT "Unit1.Em5.ControlNodes".cmCathodeNgPnpVaccum.monitoring.inWorkPos AND NOT "Unit1.Em5.ControlNodes".cmCathodeNgPnpElectrodeDetect.monitoring.processValue;
   "Unit1.Em5.ControlNodes".ngPnP.preOperationCheck.partDetect := #_w1 AND "Unit1.Em5.ControlNodes".cmCathodeNgPnpVaccum.monitoring.inWorkPos AND ("Unit1.Em5.ControlNodes".cmCathodeNgPnpElectrodeDetect.monitoring.processValue OR "Unit1.Em5.ControlNodes".cmCathodeNgPnpVaccum.monitoring.inWorkPos);
END_REGION

REGION Network 55: Gauge RnR Common Select Job
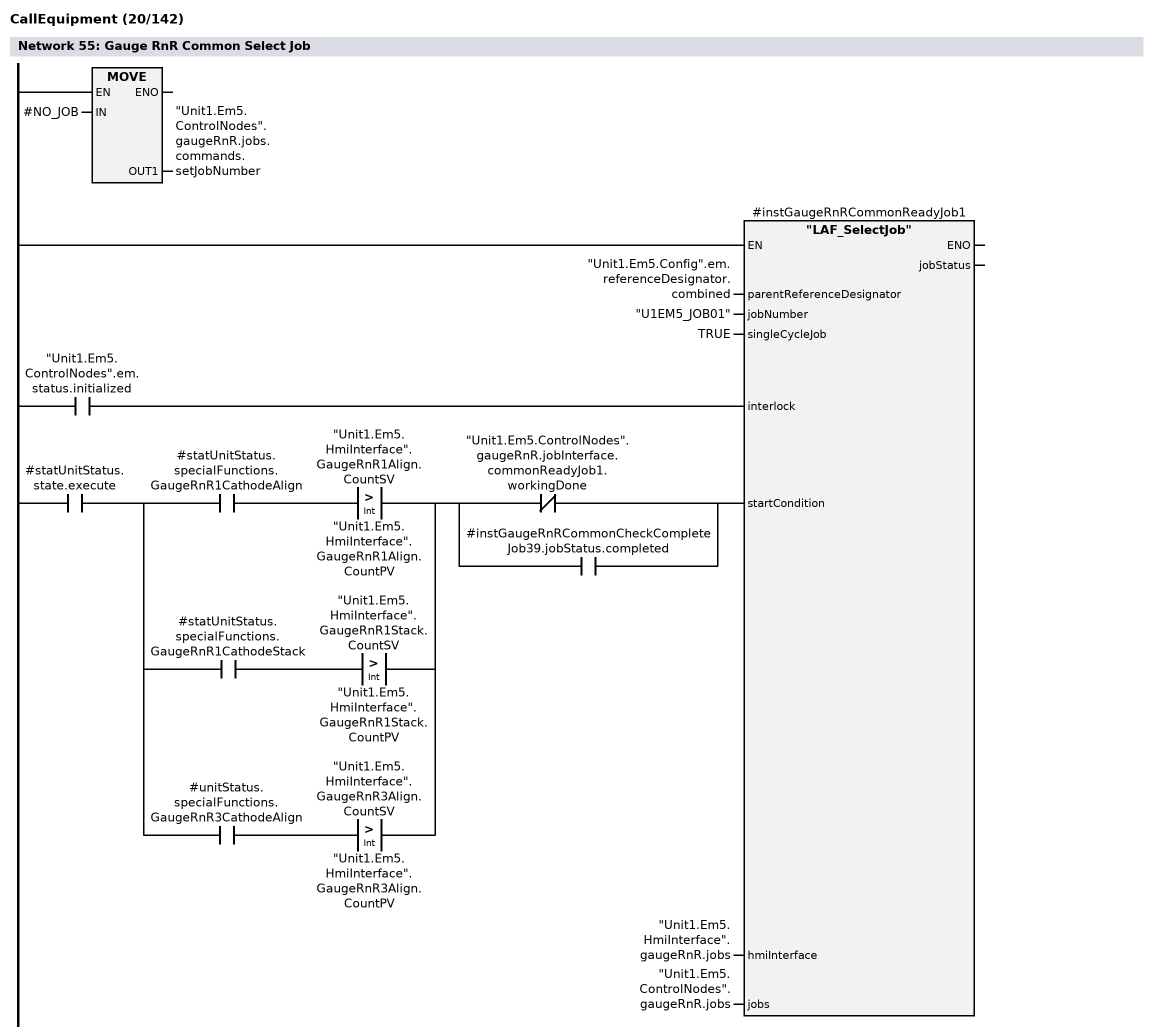
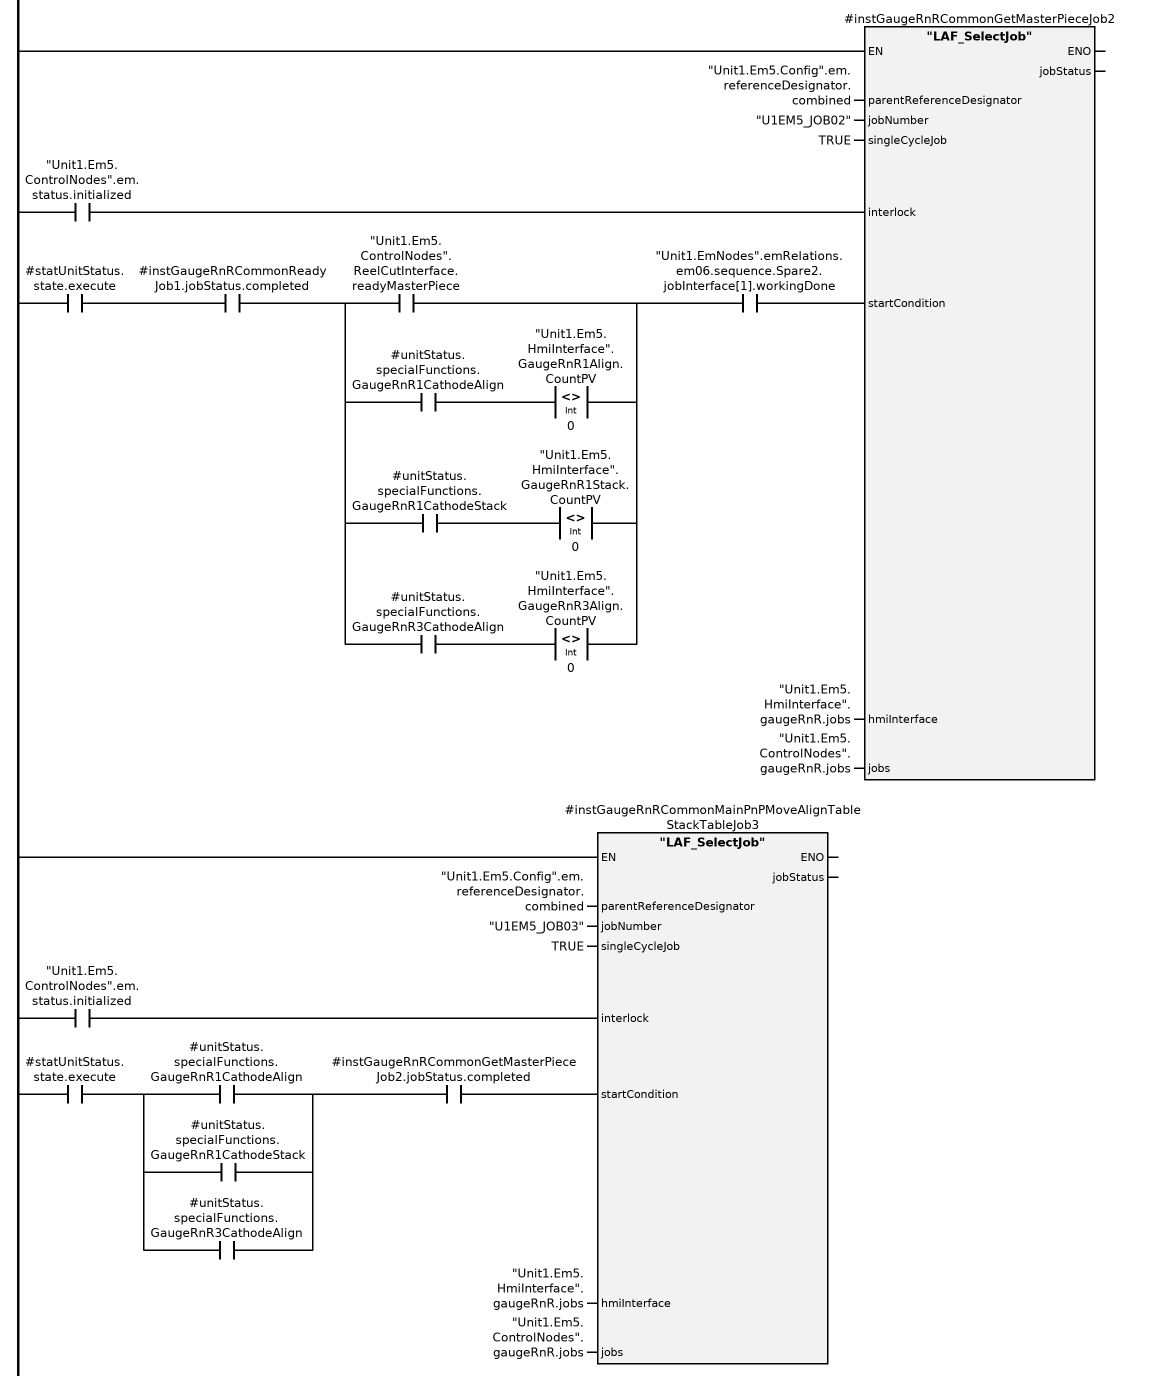
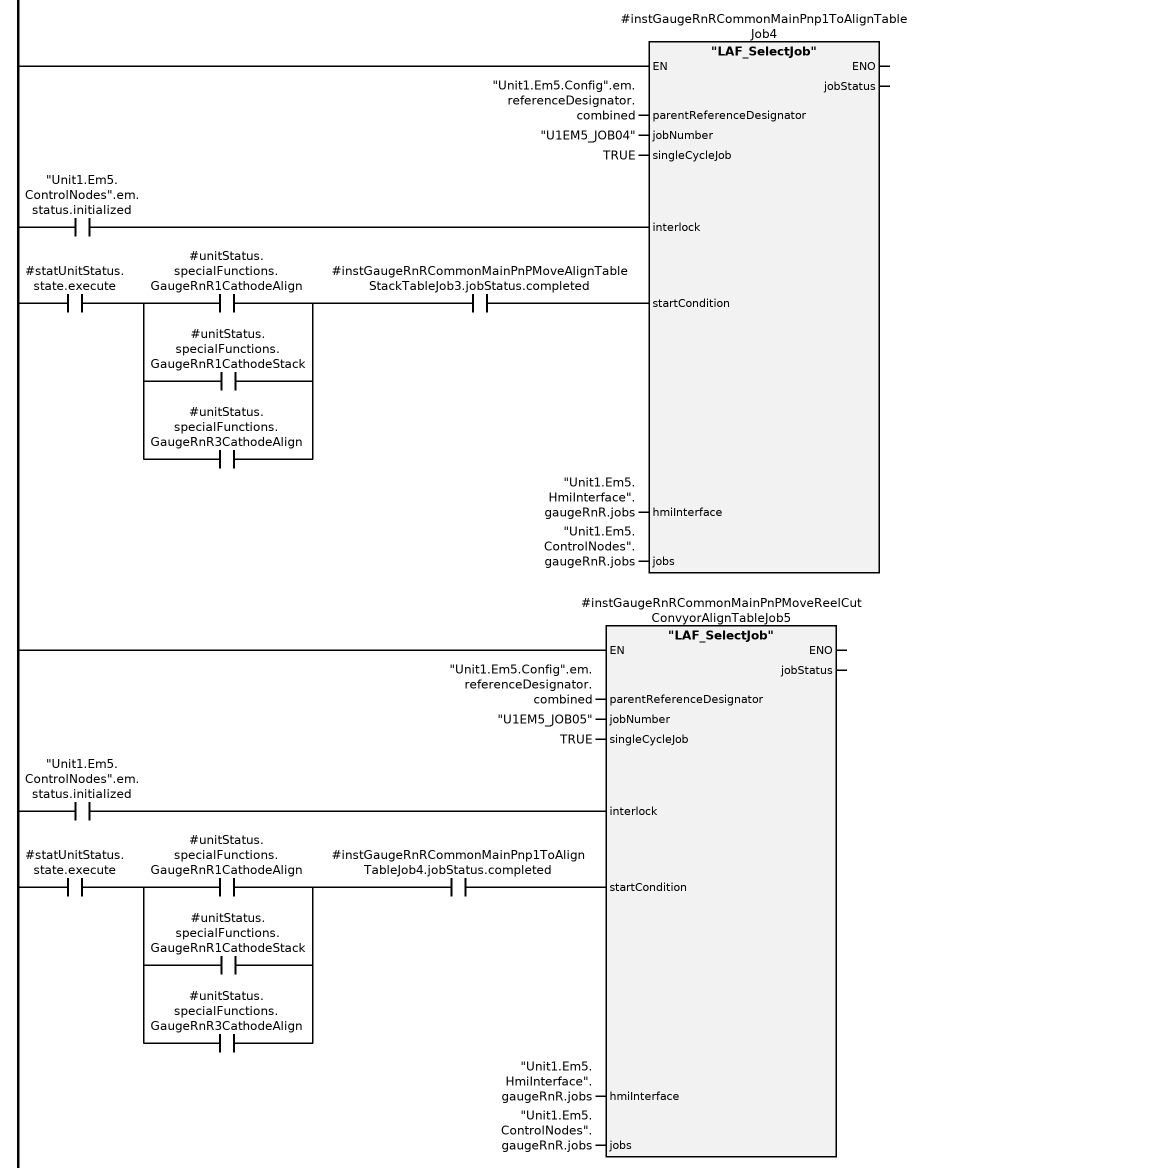
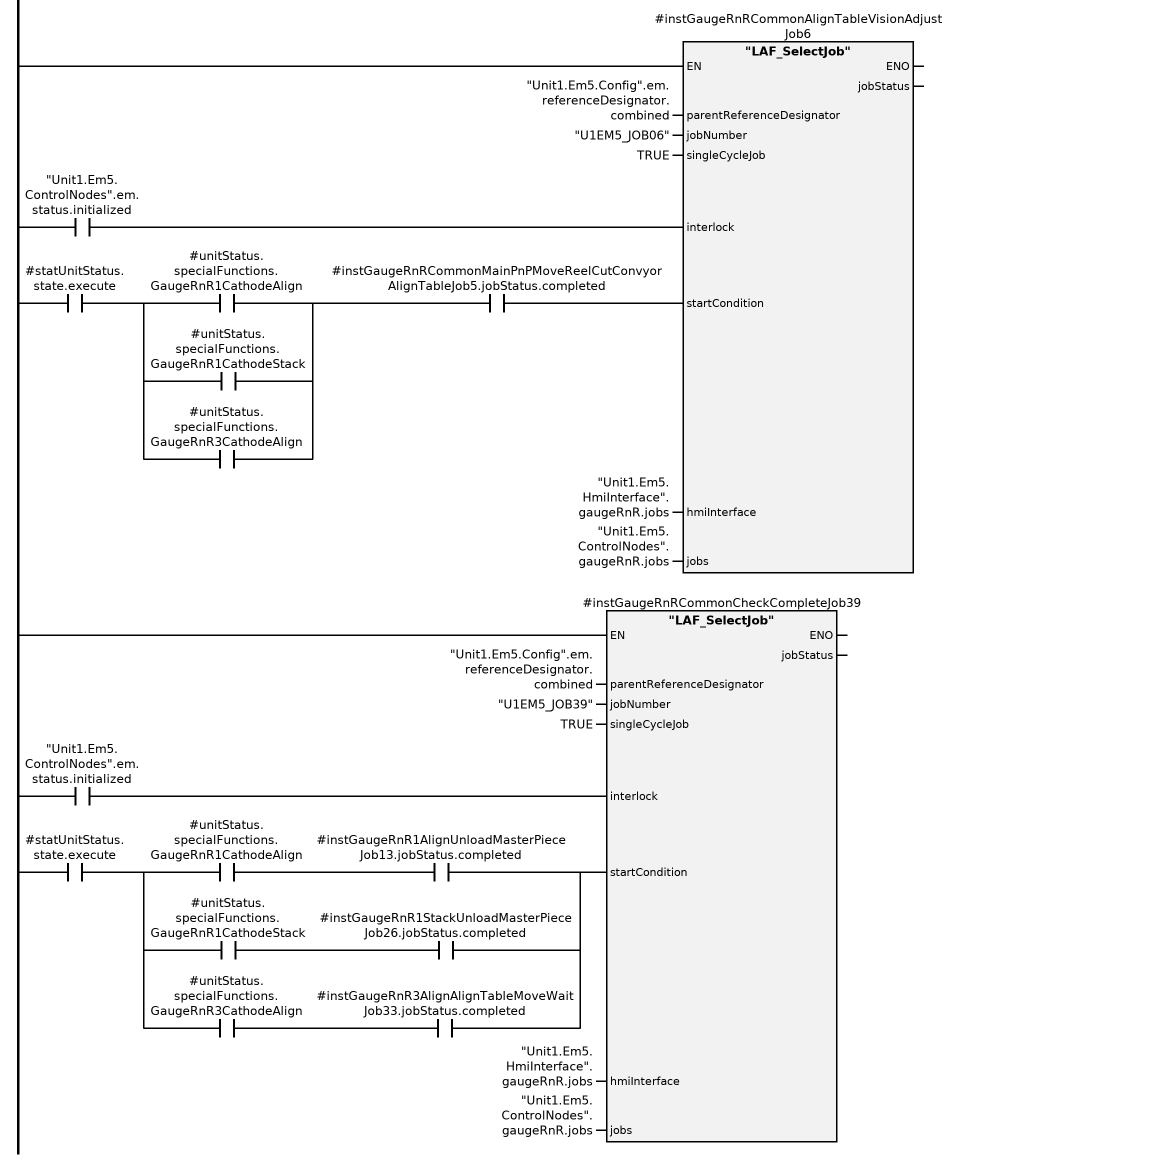
   RUNG wire#powerrail
      Move(in := #NO_JOB, out1 => "Unit1.Em5.ControlNodes".gaugeRnR.jobs.commands.setJobNumber)
   END_RUNG
   RUNG wire#powerrail
      #instGaugeRnRCommonReadyJob1(interlock := wire#w1, startCondition := wire#w4, parentReferenceDesignator := "Unit1.Em5.Config".em.referenceDesignator.combined, jobNumber := "U1EM5_JOB01", singleCycleJob := TRUE, hmiInterface := "Unit1.Em5.HmiInterface".gaugeRnR.jobs, jobs := "Unit1.Em5.ControlNodes".gaugeRnR.jobs, jobStatus =>)
   END_RUNG
   RUNG wire#powerrail
      Contact( "Unit1.Em5.ControlNodes".em.status.initialized )
   END_RUNG wire#w1
   RUNG wire#powerrail
      Contact( #statUnitStatus.state.execute )
      wire#w2
      Contact( #statUnitStatus.specialFunctions.GaugeRnR1CathodeAlign )
      { S7_Templates := "SrcType := Int" } GT_Contact(in1 := "Unit1.Em5.HmiInterface".GaugeRnR1Align.CountSV, in2 := "Unit1.Em5.HmiInterface".GaugeRnR1Align.CountPV)
      wire#w3
      I_Contact( "Unit1.Em5.ControlNodes".gaugeRnR.jobInterface.commonReadyJob1.workingDone )
   END_RUNG wire#w4
   RUNG wire#w2
      Contact( #statUnitStatus.specialFunctions.GaugeRnR1CathodeStack )
      { S7_Templates := "SrcType := Int" } GT_Contact(in1 := "Unit1.Em5.HmiInterface".GaugeRnR1Stack.CountSV, in2 := "Unit1.Em5.HmiInterface".GaugeRnR1Stack.CountPV)
   END_RUNG wire#w3
   RUNG wire#w2
      Contact( #unitStatus.specialFunctions.GaugeRnR3CathodeAlign )
      { S7_Templates := "SrcType := Int" } GT_Contact(in1 := "Unit1.Em5.HmiInterface".GaugeRnR3Align.CountSV, in2 := "Unit1.Em5.HmiInterface".GaugeRnR3Align.CountPV)
   END_RUNG wire#w3
   RUNG wire#w3
      Contact( #instGaugeRnRCommonCheckCompleteJob39.jobStatus.completed )
   END_RUNG wire#w4
   RUNG wire#powerrail
      #instGaugeRnRCommonGetMasterPieceJob2(interlock := wire#w5, startCondition := wire#w8, parentReferenceDesignator := "Unit1.Em5.Config".em.referenceDesignator.combined, jobNumber := "U1EM5_JOB02", singleCycleJob := TRUE, hmiInterface := "Unit1.Em5.HmiInterface".gaugeRnR.jobs, jobs := "Unit1.Em5.ControlNodes".gaugeRnR.jobs, jobStatus =>)
   END_RUNG
   RUNG wire#powerrail
      Contact( "Unit1.Em5.ControlNodes".em.status.initialized )
   END_RUNG wire#w5
   RUNG wire#powerrail
      Contact( #statUnitStatus.state.execute )
      Contact( #instGaugeRnRCommonReadyJob1.jobStatus.completed )
      wire#w6
      Contact( "Unit1.Em5.ControlNodes".ReelCutInterface.readyMasterPiece )
      wire#w7
      Contact( "Unit1.EmNodes".emRelations.em06.sequence.Spare2.jobInterface[1].workingDone )
   END_RUNG wire#w8
   RUNG wire#w6
      Contact( #unitStatus.specialFunctions.GaugeRnR1CathodeAlign )
      { S7_Templates := "SrcType := Int" } NE_Contact(in1 := "Unit1.Em5.HmiInterface".GaugeRnR1Align.CountPV, in2 := 0)
   END_RUNG wire#w7
   RUNG wire#w6
      Contact( #unitStatus.specialFunctions.GaugeRnR1CathodeStack )
      { S7_Templates := "SrcType := Int" } NE_Contact(in1 := "Unit1.Em5.HmiInterface".GaugeRnR1Stack.CountPV, in2 := 0)
   END_RUNG wire#w7
   RUNG wire#w6
      Contact( #unitStatus.specialFunctions.GaugeRnR3CathodeAlign )
      { S7_Templates := "SrcType := Int" } NE_Contact(in1 := "Unit1.Em5.HmiInterface".GaugeRnR3Align.CountPV, in2 := 0)
   END_RUNG wire#w7
   RUNG wire#powerrail
      #instGaugeRnRCommonMainPnPMoveAlignTableStackTableJob3(interlock := wire#w9, startCondition := wire#w12, parentReferenceDesignator := "Unit1.Em5.Config".em.referenceDesignator.combined, jobNumber := "U1EM5_JOB03", singleCycleJob := TRUE, hmiInterface := "Unit1.Em5.HmiInterface".gaugeRnR.jobs, jobs := "Unit1.Em5.ControlNodes".gaugeRnR.jobs, jobStatus =>)
   END_RUNG
   RUNG wire#powerrail
      Contact( "Unit1.Em5.ControlNodes".em.status.initialized )
   END_RUNG wire#w9
   RUNG wire#powerrail
      Contact( #statUnitStatus.state.execute )
      wire#w10
      Contact( #unitStatus.specialFunctions.GaugeRnR1CathodeAlign )
      wire#w11
      Contact( #instGaugeRnRCommonGetMasterPieceJob2.jobStatus.completed )
   END_RUNG wire#w12
   RUNG wire#w10
      Contact( #unitStatus.specialFunctions.GaugeRnR1CathodeStack )
   END_RUNG wire#w11
   RUNG wire#w10
      Contact( #unitStatus.specialFunctions.GaugeRnR3CathodeAlign )
   END_RUNG wire#w11
   RUNG wire#powerrail
      #instGaugeRnRCommonMainPnp1ToAlignTableJob4(interlock := wire#w13, startCondition := wire#w16, parentReferenceDesignator := "Unit1.Em5.Config".em.referenceDesignator.combined, jobNumber := "U1EM5_JOB04", singleCycleJob := TRUE, hmiInterface := "Unit1.Em5.HmiInterface".gaugeRnR.jobs, jobs := "Unit1.Em5.ControlNodes".gaugeRnR.jobs, jobStatus =>)
   END_RUNG
   RUNG wire#powerrail
      Contact( "Unit1.Em5.ControlNodes".em.status.initialized )
   END_RUNG wire#w13
   RUNG wire#powerrail
      Contact( #statUnitStatus.state.execute )
      wire#w14
      Contact( #unitStatus.specialFunctions.GaugeRnR1CathodeAlign )
      wire#w15
      Contact( #instGaugeRnRCommonMainPnPMoveAlignTableStackTableJob3.jobStatus.completed )
   END_RUNG wire#w16
   RUNG wire#w14
      Contact( #unitStatus.specialFunctions.GaugeRnR1CathodeStack )
   END_RUNG wire#w15
   RUNG wire#w14
      Contact( #unitStatus.specialFunctions.GaugeRnR3CathodeAlign )
   END_RUNG wire#w15
   RUNG wire#powerrail
      #instGaugeRnRCommonMainPnPMoveReelCutConvyorAlignTableJob5(interlock := wire#w17, startCondition := wire#w20, parentReferenceDesignator := "Unit1.Em5.Config".em.referenceDesignator.combined, jobNumber := "U1EM5_JOB05", singleCycleJob := TRUE, hmiInterface := "Unit1.Em5.HmiInterface".gaugeRnR.jobs, jobs := "Unit1.Em5.ControlNodes".gaugeRnR.jobs, jobStatus =>)
   END_RUNG
   RUNG wire#powerrail
      Contact( "Unit1.Em5.ControlNodes".em.status.initialized )
   END_RUNG wire#w17
   RUNG wire#powerrail
      Contact( #statUnitStatus.state.execute )
      wire#w18
      Contact( #unitStatus.specialFunctions.GaugeRnR1CathodeAlign )
      wire#w19
      Contact( #instGaugeRnRCommonMainPnp1ToAlignTableJob4.jobStatus.completed )
   END_RUNG wire#w20
   RUNG wire#w18
      Contact( #unitStatus.specialFunctions.GaugeRnR1CathodeStack )
   END_RUNG wire#w19
   RUNG wire#w18
      Contact( #unitStatus.specialFunctions.GaugeRnR3CathodeAlign )
   END_RUNG wire#w19
   RUNG wire#powerrail
      #instGaugeRnRCommonAlignTableVisionAdjustJob6(interlock := wire#w21, startCondition := wire#w24, parentReferenceDesignator := "Unit1.Em5.Config".em.referenceDesignator.combined, jobNumber := "U1EM5_JOB06", singleCycleJob := TRUE, hmiInterface := "Unit1.Em5.HmiInterface".gaugeRnR.jobs, jobs := "Unit1.Em5.ControlNodes".gaugeRnR.jobs, jobStatus =>)
   END_RUNG
   RUNG wire#powerrail
      Contact( "Unit1.Em5.ControlNodes".em.status.initialized )
   END_RUNG wire#w21
   RUNG wire#powerrail
      Contact( #statUnitStatus.state.execute )
      wire#w22
      Contact( #unitStatus.specialFunctions.GaugeRnR1CathodeAlign )
      wire#w23
      Contact( #instGaugeRnRCommonMainPnPMoveReelCutConvyorAlignTableJob5.jobStatus.completed )
   END_RUNG wire#w24
   RUNG wire#w22
      Contact( #unitStatus.specialFunctions.GaugeRnR1CathodeStack )
   END_RUNG wire#w23
   RUNG wire#w22
      Contact( #unitStatus.specialFunctions.GaugeRnR3CathodeAlign )
   END_RUNG wire#w23
   RUNG wire#powerrail
      #instGaugeRnRCommonCheckCompleteJob39(interlock := wire#w25, startCondition := wire#w27, parentReferenceDesignator := "Unit1.Em5.Config".em.referenceDesignator.combined, jobNumber := "U1EM5_JOB39", singleCycleJob := TRUE, hmiInterface := "Unit1.Em5.HmiInterface".gaugeRnR.jobs, jobs := "Unit1.Em5.ControlNodes".gaugeRnR.jobs, jobStatus =>)
   END_RUNG
   RUNG wire#powerrail
      Contact( "Unit1.Em5.ControlNodes".em.status.initialized )
   END_RUNG wire#w25
   RUNG wire#powerrail
      Contact( #statUnitStatus.state.execute )
      wire#w26
      Contact( #unitStatus.specialFunctions.GaugeRnR1CathodeAlign )
      Contact( #instGaugeRnR1AlignUnloadMasterPieceJob13.jobStatus.completed )
   END_RUNG wire#w27
   RUNG wire#w26
      Contact( #unitStatus.specialFunctions.GaugeRnR1CathodeStack )
      Contact( #instGaugeRnR1StackUnloadMasterPieceJob26.jobStatus.completed )
   END_RUNG wire#w27
   RUNG wire#w26
      Contact( #unitStatus.specialFunctions.GaugeRnR3CathodeAlign )
      Contact( #instGaugeRnR3AlignAlignTableMoveWaitJob33.jobStatus.completed )
   END_RUNG wire#w27
   // the same network as SCL:
   "Unit1.Em5.ControlNodes".gaugeRnR.jobs.commands.setJobNumber := #NO_JOB;
   #instGaugeRnRCommonReadyJob1(parentReferenceDesignator := "Unit1.Em5.Config".em.referenceDesignator.combined,   // "LAF_SelectJob"
                           jobNumber := "U1EM5_JOB01",
                           singleCycleJob := TRUE,
                           interlock := "Unit1.Em5.ControlNodes".em.status.initialized,
                           startCondition := #statUnitStatus.state.execute AND ((#statUnitStatus.specialFunctions.GaugeRnR1CathodeAlign AND ("Unit1.Em5.HmiInterface".GaugeRnR1Align.CountSV > "Unit1.Em5.HmiInterface".GaugeRnR1Align.CountPV)) OR (#statUnitStatus.specialFunctions.GaugeRnR1CathodeStack AND ("Unit1.Em5.HmiInterface".GaugeRnR1Stack.CountSV > "Unit1.Em5.HmiInterface".GaugeRnR1Stack.CountPV)) OR (#unitStatus.specialFunctions.GaugeRnR3CathodeAlign AND ("Unit1.Em5.HmiInterface".GaugeRnR3Align.CountSV > "Unit1.Em5.HmiInterface".GaugeRnR3Align.CountPV))) AND (NOT "Unit1.Em5.ControlNodes".gaugeRnR.jobInterface.commonReadyJob1.workingDone OR #instGaugeRnRCommonCheckCompleteJob39.jobStatus.completed),
                           hmiInterface := "Unit1.Em5.HmiInterface".gaugeRnR.jobs,
                           jobs := "Unit1.Em5.ControlNodes".gaugeRnR.jobs);
   #instGaugeRnRCommonGetMasterPieceJob2(parentReferenceDesignator := "Unit1.Em5.Config".em.referenceDesignator.combined,   // "LAF_SelectJob"
                           jobNumber := "U1EM5_JOB02",
                           singleCycleJob := TRUE,
                           interlock := "Unit1.Em5.ControlNodes".em.status.initialized,
                           startCondition := #statUnitStatus.state.execute AND #instGaugeRnRCommonReadyJob1.jobStatus.completed AND ("Unit1.Em5.ControlNodes".ReelCutInterface.readyMasterPiece OR (#unitStatus.specialFunctions.GaugeRnR1CathodeAlign AND ("Unit1.Em5.HmiInterface".GaugeRnR1Align.CountPV <> 0)) OR (#unitStatus.specialFunctions.GaugeRnR1CathodeStack AND ("Unit1.Em5.HmiInterface".GaugeRnR1Stack.CountPV <> 0)) OR (#unitStatus.specialFunctions.GaugeRnR3CathodeAlign AND ("Unit1.Em5.HmiInterface".GaugeRnR3Align.CountPV <> 0))) AND "Unit1.EmNodes".emRelations.em06.sequence.Spare2.jobInterface[1].workingDone,
                           hmiInterface := "Unit1.Em5.HmiInterface".gaugeRnR.jobs,
                           jobs := "Unit1.Em5.ControlNodes".gaugeRnR.jobs);
   #instGaugeRnRCommonMainPnPMoveAlignTableStackTableJob3(parentReferenceDesignator := "Unit1.Em5.Config".em.referenceDesignator.combined,   // "LAF_SelectJob"
                           jobNumber := "U1EM5_JOB03",
                           singleCycleJob := TRUE,
                           interlock := "Unit1.Em5.ControlNodes".em.status.initialized,
                           startCondition := #statUnitStatus.state.execute AND (#unitStatus.specialFunctions.GaugeRnR1CathodeAlign OR #unitStatus.specialFunctions.GaugeRnR1CathodeStack OR #unitStatus.specialFunctions.GaugeRnR3CathodeAlign) AND #instGaugeRnRCommonGetMasterPieceJob2.jobStatus.completed,
                           hmiInterface := "Unit1.Em5.HmiInterface".gaugeRnR.jobs,
                           jobs := "Unit1.Em5.ControlNodes".gaugeRnR.jobs);
   #instGaugeRnRCommonMainPnp1ToAlignTableJob4(parentReferenceDesignator := "Unit1.Em5.Config".em.referenceDesignator.combined,   // "LAF_SelectJob"
                           jobNumber := "U1EM5_JOB04",
                           singleCycleJob := TRUE,
                           interlock := "Unit1.Em5.ControlNodes".em.status.initialized,
                           startCondition := #statUnitStatus.state.execute AND (#unitStatus.specialFunctions.GaugeRnR1CathodeAlign OR #unitStatus.specialFunctions.GaugeRnR1CathodeStack OR #unitStatus.specialFunctions.GaugeRnR3CathodeAlign) AND #instGaugeRnRCommonMainPnPMoveAlignTableStackTableJob3.jobStatus.completed,
                           hmiInterface := "Unit1.Em5.HmiInterface".gaugeRnR.jobs,
                           jobs := "Unit1.Em5.ControlNodes".gaugeRnR.jobs);
   #instGaugeRnRCommonMainPnPMoveReelCutConvyorAlignTableJob5(parentReferenceDesignator := "Unit1.Em5.Config".em.referenceDesignator.combined,   // "LAF_SelectJob"
                           jobNumber := "U1EM5_JOB05",
                           singleCycleJob := TRUE,
                           interlock := "Unit1.Em5.ControlNodes".em.status.initialized,
                           startCondition := #statUnitStatus.state.execute AND (#unitStatus.specialFunctions.GaugeRnR1CathodeAlign OR #unitStatus.specialFunctions.GaugeRnR1CathodeStack OR #unitStatus.specialFunctions.GaugeRnR3CathodeAlign) AND #instGaugeRnRCommonMainPnp1ToAlignTableJob4.jobStatus.completed,
                           hmiInterface := "Unit1.Em5.HmiInterface".gaugeRnR.jobs,
                           jobs := "Unit1.Em5.ControlNodes".gaugeRnR.jobs);
   #instGaugeRnRCommonAlignTableVisionAdjustJob6(parentReferenceDesignator := "Unit1.Em5.Config".em.referenceDesignator.combined,   // "LAF_SelectJob"
                           jobNumber := "U1EM5_JOB06",
                           singleCycleJob := TRUE,
                           interlock := "Unit1.Em5.ControlNodes".em.status.initialized,
                           startCondition := #statUnitStatus.state.execute AND (#unitStatus.specialFunctions.GaugeRnR1CathodeAlign OR #unitStatus.specialFunctions.GaugeRnR1CathodeStack OR #unitStatus.specialFunctions.GaugeRnR3CathodeAlign) AND #instGaugeRnRCommonMainPnPMoveReelCutConvyorAlignTableJob5.jobStatus.completed,
                           hmiInterface := "Unit1.Em5.HmiInterface".gaugeRnR.jobs,
                           jobs := "Unit1.Em5.ControlNodes".gaugeRnR.jobs);
   #instGaugeRnRCommonCheckCompleteJob39(parentReferenceDesignator := "Unit1.Em5.Config".em.referenceDesignator.combined,   // "LAF_SelectJob"
                           jobNumber := "U1EM5_JOB39",
                           singleCycleJob := TRUE,
                           interlock := "Unit1.Em5.ControlNodes".em.status.initialized,
                           startCondition := #statUnitStatus.state.execute AND ((#unitStatus.specialFunctions.GaugeRnR1CathodeAlign AND #instGaugeRnR1AlignUnloadMasterPieceJob13.jobStatus.completed) OR (#unitStatus.specialFunctions.GaugeRnR1CathodeStack AND #instGaugeRnR1StackUnloadMasterPieceJob26.jobStatus.completed) OR (#unitStatus.specialFunctions.GaugeRnR3CathodeAlign AND #instGaugeRnR3AlignAlignTableMoveWaitJob33.jobStatus.completed)),
                           hmiInterface := "Unit1.Em5.HmiInterface".gaugeRnR.jobs,
                           jobs := "Unit1.Em5.ControlNodes".gaugeRnR.jobs);
END_REGION

REGION Network 56: Gauge RnR 1 Align Select Job
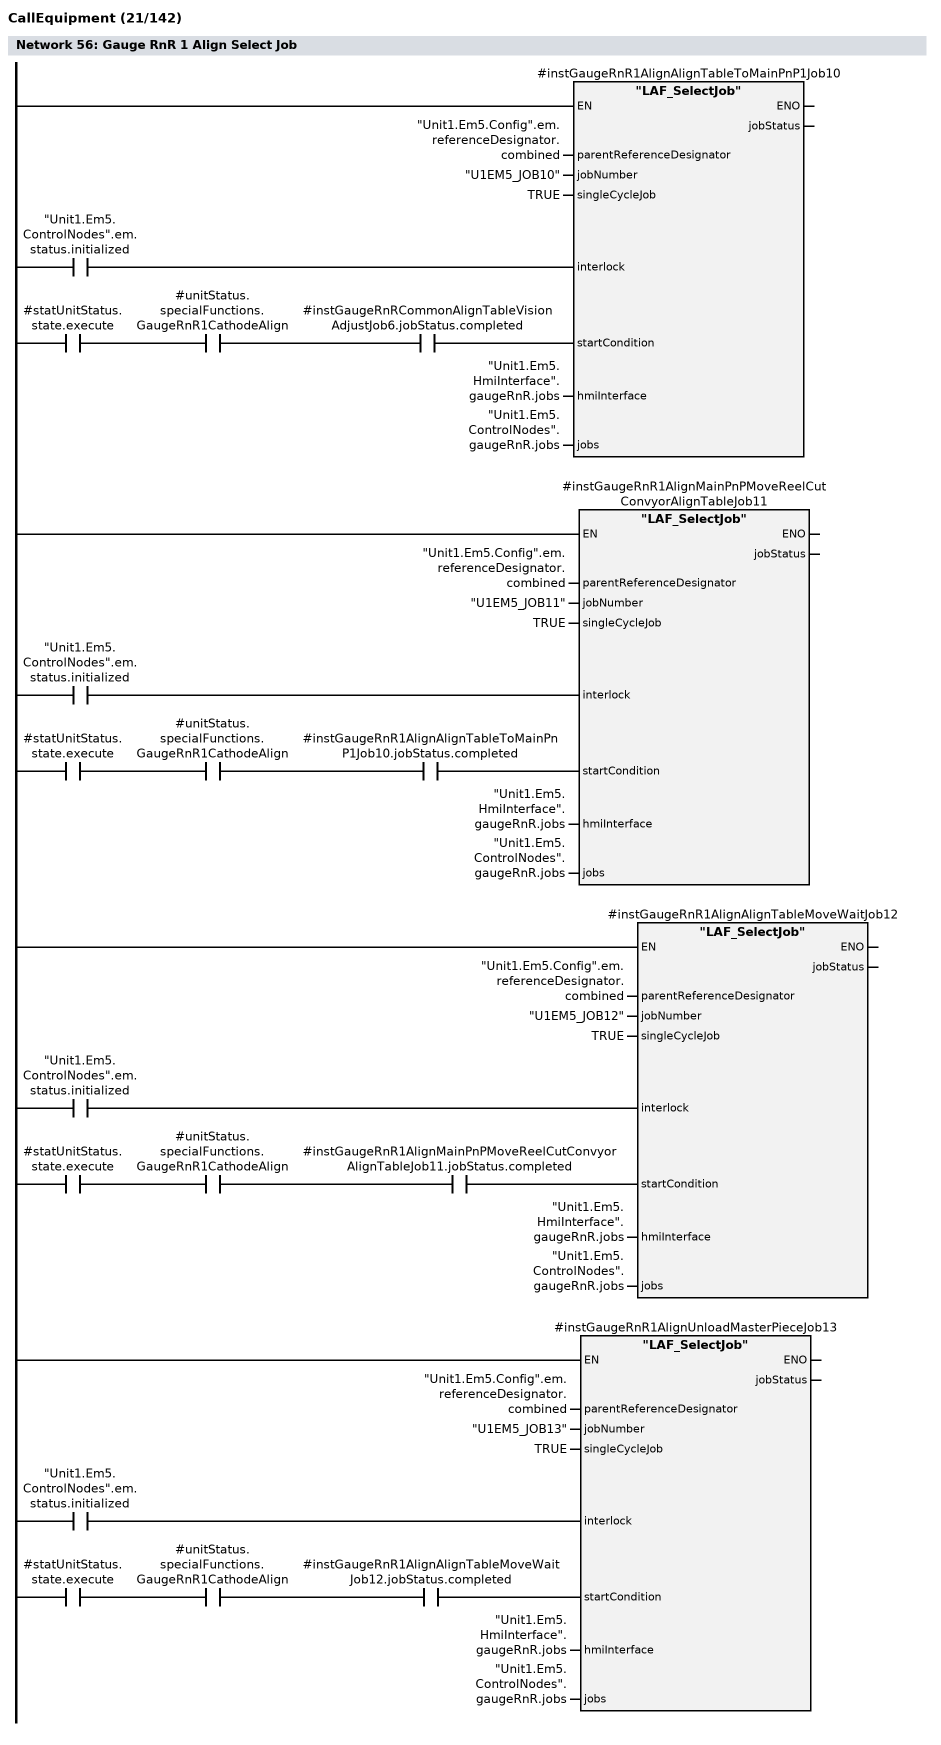
   RUNG wire#powerrail
      #instGaugeRnR1AlignAlignTableToMainPnP1Job10(interlock := wire#w1, startCondition := wire#w2, parentReferenceDesignator := "Unit1.Em5.Config".em.referenceDesignator.combined, jobNumber := "U1EM5_JOB10", singleCycleJob := TRUE, hmiInterface := "Unit1.Em5.HmiInterface".gaugeRnR.jobs, jobs := "Unit1.Em5.ControlNodes".gaugeRnR.jobs, jobStatus =>)
   END_RUNG
   RUNG wire#powerrail
      Contact( "Unit1.Em5.ControlNodes".em.status.initialized )
   END_RUNG wire#w1
   RUNG wire#powerrail
      Contact( #statUnitStatus.state.execute )
      Contact( #unitStatus.specialFunctions.GaugeRnR1CathodeAlign )
      Contact( #instGaugeRnRCommonAlignTableVisionAdjustJob6.jobStatus.completed )
   END_RUNG wire#w2
   RUNG wire#powerrail
      #instGaugeRnR1AlignMainPnPMoveReelCutConvyorAlignTableJob11(interlock := wire#w3, startCondition := wire#w4, parentReferenceDesignator := "Unit1.Em5.Config".em.referenceDesignator.combined, jobNumber := "U1EM5_JOB11", singleCycleJob := TRUE, hmiInterface := "Unit1.Em5.HmiInterface".gaugeRnR.jobs, jobs := "Unit1.Em5.ControlNodes".gaugeRnR.jobs, jobStatus =>)
   END_RUNG
   RUNG wire#powerrail
      Contact( "Unit1.Em5.ControlNodes".em.status.initialized )
   END_RUNG wire#w3
   RUNG wire#powerrail
      Contact( #statUnitStatus.state.execute )
      Contact( #unitStatus.specialFunctions.GaugeRnR1CathodeAlign )
      Contact( #instGaugeRnR1AlignAlignTableToMainPnP1Job10.jobStatus.completed )
   END_RUNG wire#w4
   RUNG wire#powerrail
      #instGaugeRnR1AlignAlignTableMoveWaitJob12(interlock := wire#w5, startCondition := wire#w6, parentReferenceDesignator := "Unit1.Em5.Config".em.referenceDesignator.combined, jobNumber := "U1EM5_JOB12", singleCycleJob := TRUE, hmiInterface := "Unit1.Em5.HmiInterface".gaugeRnR.jobs, jobs := "Unit1.Em5.ControlNodes".gaugeRnR.jobs, jobStatus =>)
   END_RUNG
   RUNG wire#powerrail
      Contact( "Unit1.Em5.ControlNodes".em.status.initialized )
   END_RUNG wire#w5
   RUNG wire#powerrail
      Contact( #statUnitStatus.state.execute )
      Contact( #unitStatus.specialFunctions.GaugeRnR1CathodeAlign )
      Contact( #instGaugeRnR1AlignMainPnPMoveReelCutConvyorAlignTableJob11.jobStatus.completed )
   END_RUNG wire#w6
   RUNG wire#powerrail
      #instGaugeRnR1AlignUnloadMasterPieceJob13(interlock := wire#w7, startCondition := wire#w8, parentReferenceDesignator := "Unit1.Em5.Config".em.referenceDesignator.combined, jobNumber := "U1EM5_JOB13", singleCycleJob := TRUE, hmiInterface := "Unit1.Em5.HmiInterface".gaugeRnR.jobs, jobs := "Unit1.Em5.ControlNodes".gaugeRnR.jobs, jobStatus =>)
   END_RUNG
   RUNG wire#powerrail
      Contact( "Unit1.Em5.ControlNodes".em.status.initialized )
   END_RUNG wire#w7
   RUNG wire#powerrail
      Contact( #statUnitStatus.state.execute )
      Contact( #unitStatus.specialFunctions.GaugeRnR1CathodeAlign )
      Contact( #instGaugeRnR1AlignAlignTableMoveWaitJob12.jobStatus.completed )
   END_RUNG wire#w8
   // the same network as SCL:
   #instGaugeRnR1AlignAlignTableToMainPnP1Job10(parentReferenceDesignator := "Unit1.Em5.Config".em.referenceDesignator.combined,   // "LAF_SelectJob"
                           jobNumber := "U1EM5_JOB10",
                           singleCycleJob := TRUE,
                           interlock := "Unit1.Em5.ControlNodes".em.status.initialized,
                           startCondition := #statUnitStatus.state.execute AND #unitStatus.specialFunctions.GaugeRnR1CathodeAlign AND #instGaugeRnRCommonAlignTableVisionAdjustJob6.jobStatus.completed,
                           hmiInterface := "Unit1.Em5.HmiInterface".gaugeRnR.jobs,
                           jobs := "Unit1.Em5.ControlNodes".gaugeRnR.jobs);
   #instGaugeRnR1AlignMainPnPMoveReelCutConvyorAlignTableJob11(parentReferenceDesignator := "Unit1.Em5.Config".em.referenceDesignator.combined,   // "LAF_SelectJob"
                           jobNumber := "U1EM5_JOB11",
                           singleCycleJob := TRUE,
                           interlock := "Unit1.Em5.ControlNodes".em.status.initialized,
                           startCondition := #statUnitStatus.state.execute AND #unitStatus.specialFunctions.GaugeRnR1CathodeAlign AND #instGaugeRnR1AlignAlignTableToMainPnP1Job10.jobStatus.completed,
                           hmiInterface := "Unit1.Em5.HmiInterface".gaugeRnR.jobs,
                           jobs := "Unit1.Em5.ControlNodes".gaugeRnR.jobs);
   #instGaugeRnR1AlignAlignTableMoveWaitJob12(parentReferenceDesignator := "Unit1.Em5.Config".em.referenceDesignator.combined,   // "LAF_SelectJob"
                           jobNumber := "U1EM5_JOB12",
                           singleCycleJob := TRUE,
                           interlock := "Unit1.Em5.ControlNodes".em.status.initialized,
                           startCondition := #statUnitStatus.state.execute AND #unitStatus.specialFunctions.GaugeRnR1CathodeAlign AND #instGaugeRnR1AlignMainPnPMoveReelCutConvyorAlignTableJob11.jobStatus.completed,
                           hmiInterface := "Unit1.Em5.HmiInterface".gaugeRnR.jobs,
                           jobs := "Unit1.Em5.ControlNodes".gaugeRnR.jobs);
   #instGaugeRnR1AlignUnloadMasterPieceJob13(parentReferenceDesignator := "Unit1.Em5.Config".em.referenceDesignator.combined,   // "LAF_SelectJob"
                           jobNumber := "U1EM5_JOB13",
                           singleCycleJob := TRUE,
                           interlock := "Unit1.Em5.ControlNodes".em.status.initialized,
                           startCondition := #statUnitStatus.state.execute AND #unitStatus.specialFunctions.GaugeRnR1CathodeAlign AND #instGaugeRnR1AlignAlignTableMoveWaitJob12.jobStatus.completed,
                           hmiInterface := "Unit1.Em5.HmiInterface".gaugeRnR.jobs,
                           jobs := "Unit1.Em5.ControlNodes".gaugeRnR.jobs);
END_REGION

REGION Network 57: Gauge RnR 1 Stack Select Job
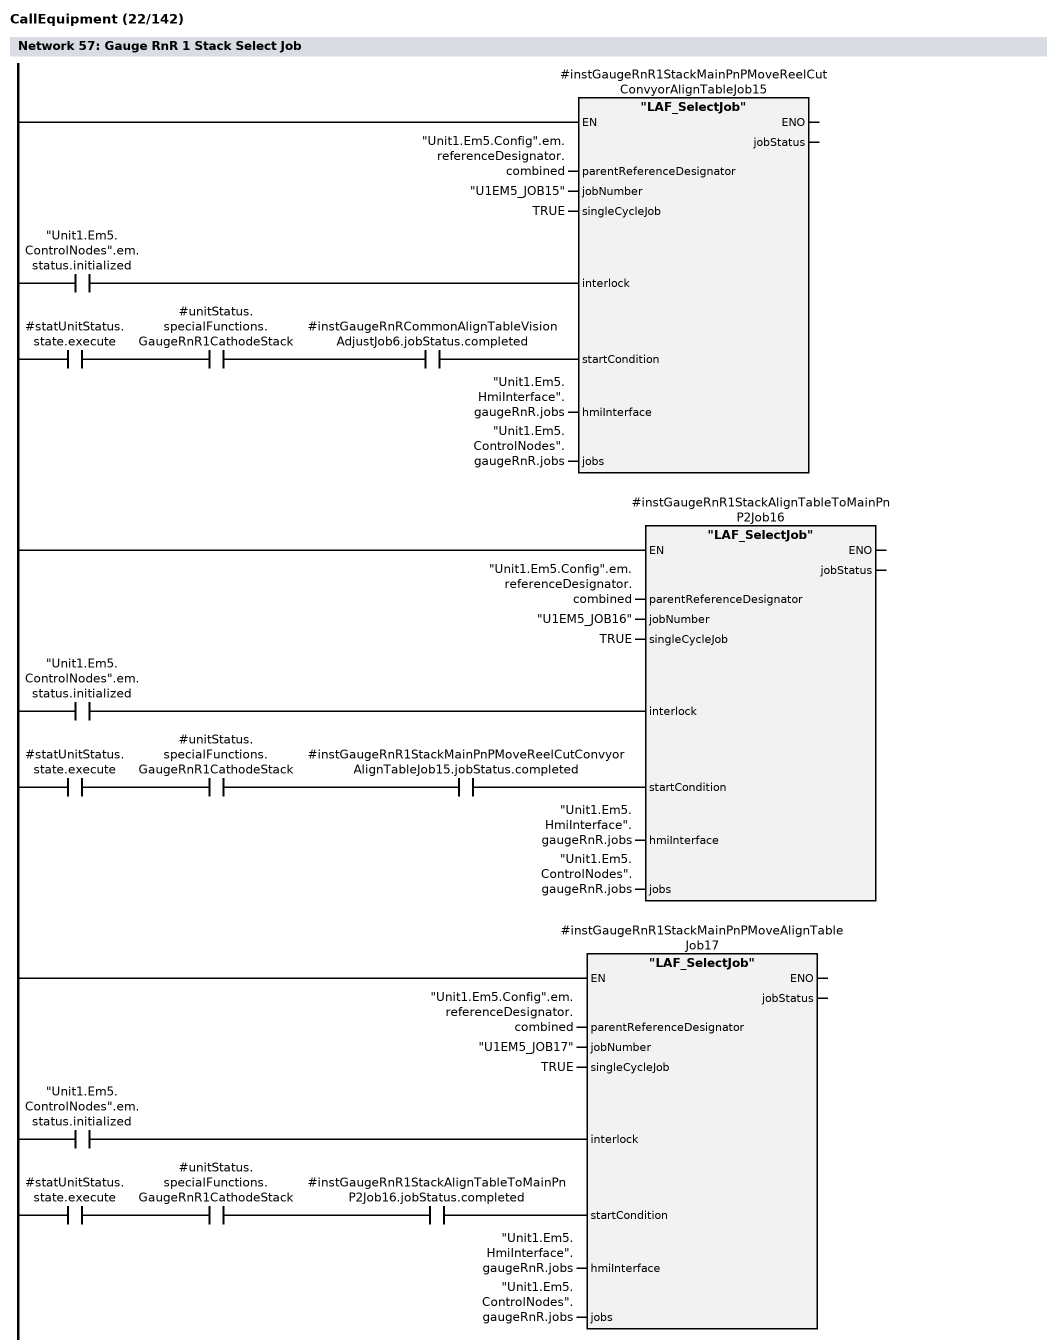
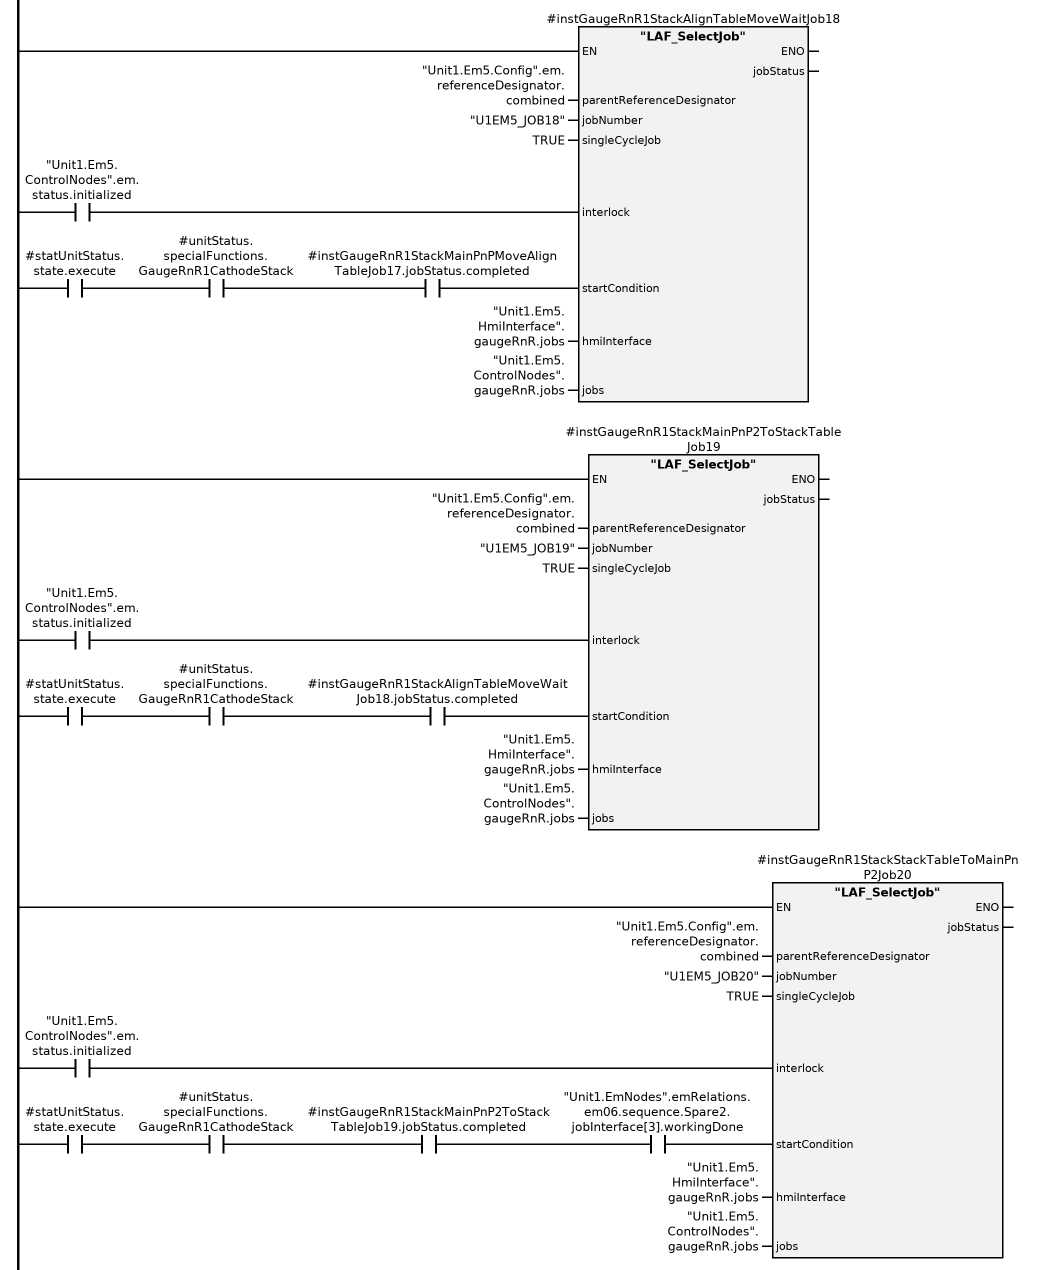
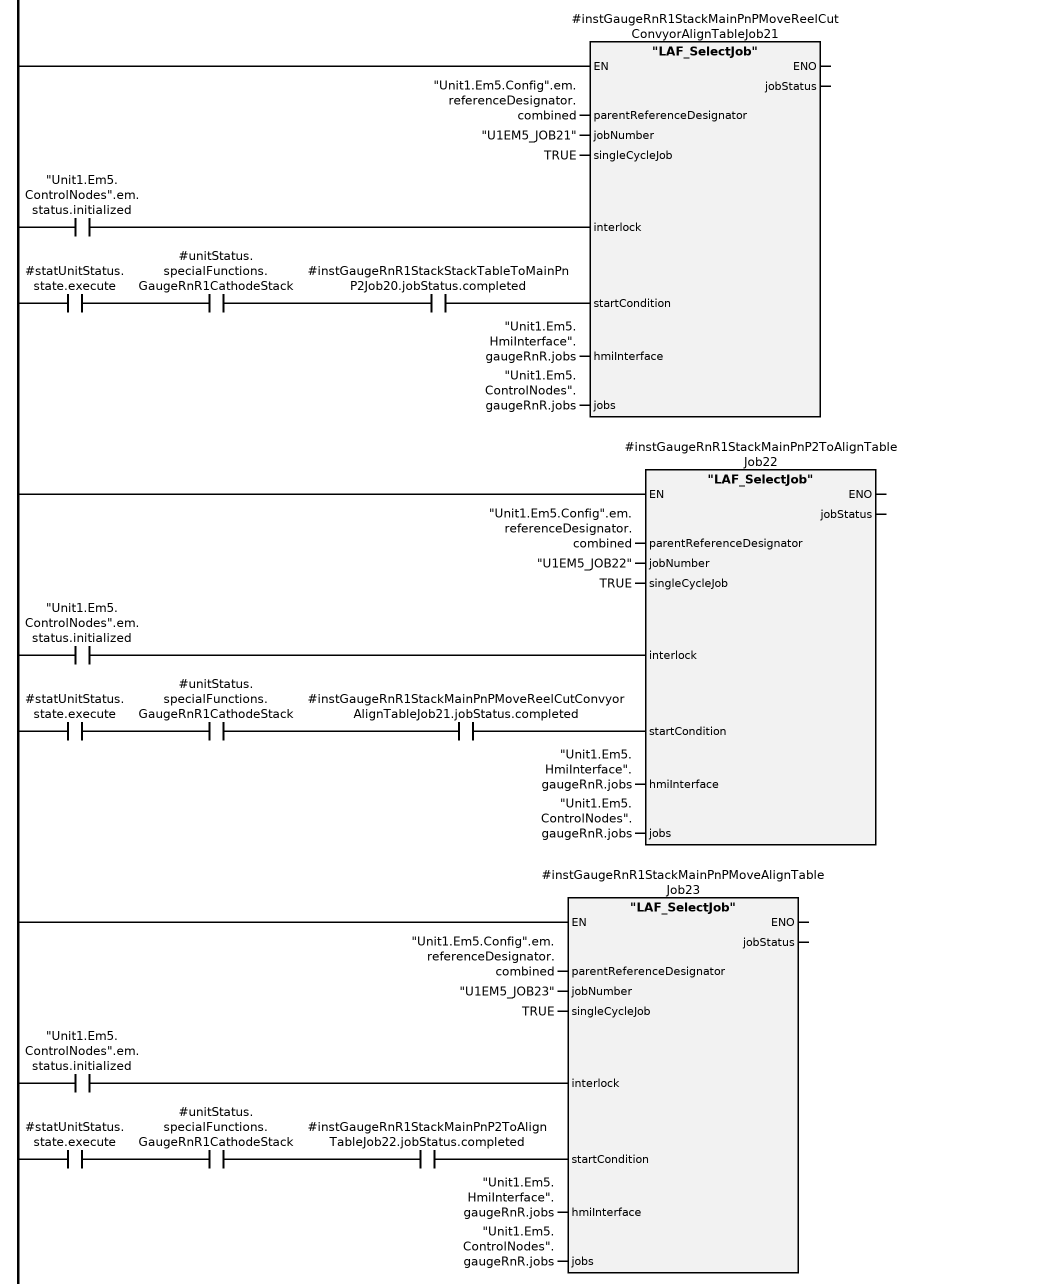
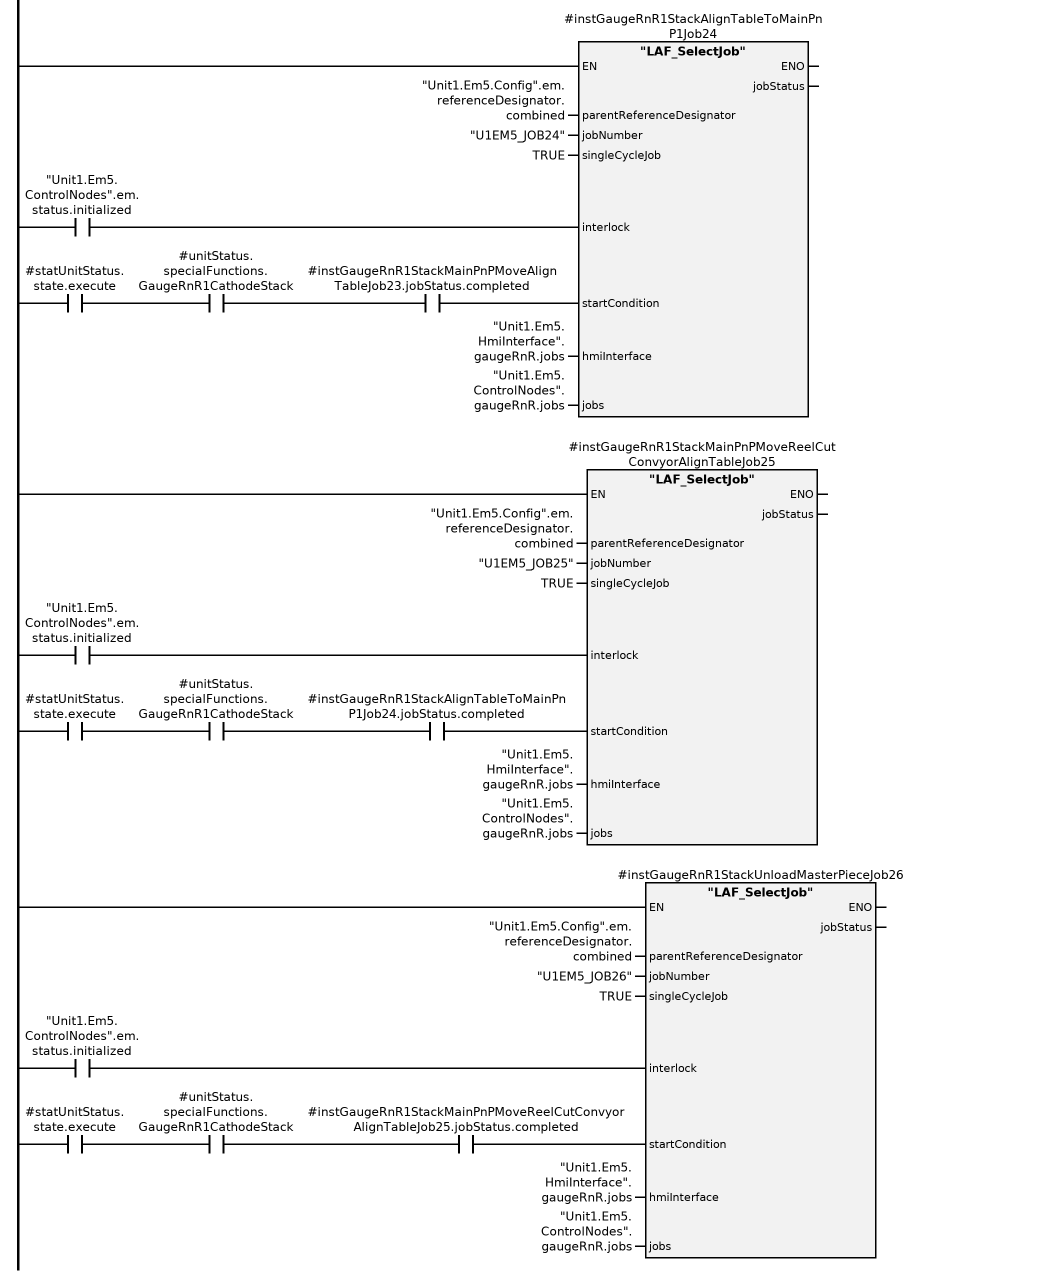
   RUNG wire#powerrail
      #instGaugeRnR1StackMainPnPMoveReelCutConvyorAlignTableJob15(interlock := wire#w1, startCondition := wire#w2, parentReferenceDesignator := "Unit1.Em5.Config".em.referenceDesignator.combined, jobNumber := "U1EM5_JOB15", singleCycleJob := TRUE, hmiInterface := "Unit1.Em5.HmiInterface".gaugeRnR.jobs, jobs := "Unit1.Em5.ControlNodes".gaugeRnR.jobs, jobStatus =>)
   END_RUNG
   RUNG wire#powerrail
      Contact( "Unit1.Em5.ControlNodes".em.status.initialized )
   END_RUNG wire#w1
   RUNG wire#powerrail
      Contact( #statUnitStatus.state.execute )
      Contact( #unitStatus.specialFunctions.GaugeRnR1CathodeStack )
      Contact( #instGaugeRnRCommonAlignTableVisionAdjustJob6.jobStatus.completed )
   END_RUNG wire#w2
   RUNG wire#powerrail
      #instGaugeRnR1StackAlignTableToMainPnP2Job16(interlock := wire#w3, startCondition := wire#w4, parentReferenceDesignator := "Unit1.Em5.Config".em.referenceDesignator.combined, jobNumber := "U1EM5_JOB16", singleCycleJob := TRUE, hmiInterface := "Unit1.Em5.HmiInterface".gaugeRnR.jobs, jobs := "Unit1.Em5.ControlNodes".gaugeRnR.jobs, jobStatus =>)
   END_RUNG
   RUNG wire#powerrail
      Contact( "Unit1.Em5.ControlNodes".em.status.initialized )
   END_RUNG wire#w3
   RUNG wire#powerrail
      Contact( #statUnitStatus.state.execute )
      Contact( #unitStatus.specialFunctions.GaugeRnR1CathodeStack )
      Contact( #instGaugeRnR1StackMainPnPMoveReelCutConvyorAlignTableJob15.jobStatus.completed )
   END_RUNG wire#w4
   RUNG wire#powerrail
      #instGaugeRnR1StackMainPnPMoveAlignTableJob17(interlock := wire#w5, startCondition := wire#w6, parentReferenceDesignator := "Unit1.Em5.Config".em.referenceDesignator.combined, jobNumber := "U1EM5_JOB17", singleCycleJob := TRUE, hmiInterface := "Unit1.Em5.HmiInterface".gaugeRnR.jobs, jobs := "Unit1.Em5.ControlNodes".gaugeRnR.jobs, jobStatus =>)
   END_RUNG
   RUNG wire#powerrail
      Contact( "Unit1.Em5.ControlNodes".em.status.initialized )
   END_RUNG wire#w5
   RUNG wire#powerrail
      Contact( #statUnitStatus.state.execute )
      Contact( #unitStatus.specialFunctions.GaugeRnR1CathodeStack )
      Contact( #instGaugeRnR1StackAlignTableToMainPnP2Job16.jobStatus.completed )
   END_RUNG wire#w6
   RUNG wire#powerrail
      #instGaugeRnR1StackAlignTableMoveWaitJob18(interlock := wire#w7, startCondition := wire#w8, parentReferenceDesignator := "Unit1.Em5.Config".em.referenceDesignator.combined, jobNumber := "U1EM5_JOB18", singleCycleJob := TRUE, hmiInterface := "Unit1.Em5.HmiInterface".gaugeRnR.jobs, jobs := "Unit1.Em5.ControlNodes".gaugeRnR.jobs, jobStatus =>)
   END_RUNG
   RUNG wire#powerrail
      Contact( "Unit1.Em5.ControlNodes".em.status.initialized )
   END_RUNG wire#w7
   RUNG wire#powerrail
      Contact( #statUnitStatus.state.execute )
      Contact( #unitStatus.specialFunctions.GaugeRnR1CathodeStack )
      Contact( #instGaugeRnR1StackMainPnPMoveAlignTableJob17.jobStatus.completed )
   END_RUNG wire#w8
   RUNG wire#powerrail
      #instGaugeRnR1StackMainPnP2ToStackTableJob19(interlock := wire#w9, startCondition := wire#w10, parentReferenceDesignator := "Unit1.Em5.Config".em.referenceDesignator.combined, jobNumber := "U1EM5_JOB19", singleCycleJob := TRUE, hmiInterface := "Unit1.Em5.HmiInterface".gaugeRnR.jobs, jobs := "Unit1.Em5.ControlNodes".gaugeRnR.jobs, jobStatus =>)
   END_RUNG
   RUNG wire#powerrail
      Contact( "Unit1.Em5.ControlNodes".em.status.initialized )
   END_RUNG wire#w9
   RUNG wire#powerrail
      Contact( #statUnitStatus.state.execute )
      Contact( #unitStatus.specialFunctions.GaugeRnR1CathodeStack )
      Contact( #instGaugeRnR1StackAlignTableMoveWaitJob18.jobStatus.completed )
   END_RUNG wire#w10
   RUNG wire#powerrail
      #instGaugeRnR1StackStackTableToMainPnP2Job20(interlock := wire#w11, startCondition := wire#w12, parentReferenceDesignator := "Unit1.Em5.Config".em.referenceDesignator.combined, jobNumber := "U1EM5_JOB20", singleCycleJob := TRUE, hmiInterface := "Unit1.Em5.HmiInterface".gaugeRnR.jobs, jobs := "Unit1.Em5.ControlNodes".gaugeRnR.jobs, jobStatus =>)
   END_RUNG
   RUNG wire#powerrail
      Contact( "Unit1.Em5.ControlNodes".em.status.initialized )
   END_RUNG wire#w11
   RUNG wire#powerrail
      Contact( #statUnitStatus.state.execute )
      Contact( #unitStatus.specialFunctions.GaugeRnR1CathodeStack )
      Contact( #instGaugeRnR1StackMainPnP2ToStackTableJob19.jobStatus.completed )
      Contact( "Unit1.EmNodes".emRelations.em06.sequence.Spare2.jobInterface[3].workingDone )
   END_RUNG wire#w12
   RUNG wire#powerrail
      #instGaugeRnR1StackMainPnPMoveReelCutConvyorAlignTableJob21(interlock := wire#w13, startCondition := wire#w14, parentReferenceDesignator := "Unit1.Em5.Config".em.referenceDesignator.combined, jobNumber := "U1EM5_JOB21", singleCycleJob := TRUE, hmiInterface := "Unit1.Em5.HmiInterface".gaugeRnR.jobs, jobs := "Unit1.Em5.ControlNodes".gaugeRnR.jobs, jobStatus =>)
   END_RUNG
   RUNG wire#powerrail
      Contact( "Unit1.Em5.ControlNodes".em.status.initialized )
   END_RUNG wire#w13
   RUNG wire#powerrail
      Contact( #statUnitStatus.state.execute )
      Contact( #unitStatus.specialFunctions.GaugeRnR1CathodeStack )
      Contact( #instGaugeRnR1StackStackTableToMainPnP2Job20.jobStatus.completed )
   END_RUNG wire#w14
   RUNG wire#powerrail
      #instGaugeRnR1StackMainPnP2ToAlignTableJob22(interlock := wire#w15, startCondition := wire#w16, parentReferenceDesignator := "Unit1.Em5.Config".em.referenceDesignator.combined, jobNumber := "U1EM5_JOB22", singleCycleJob := TRUE, hmiInterface := "Unit1.Em5.HmiInterface".gaugeRnR.jobs, jobs := "Unit1.Em5.ControlNodes".gaugeRnR.jobs, jobStatus =>)
   END_RUNG
   RUNG wire#powerrail
      Contact( "Unit1.Em5.ControlNodes".em.status.initialized )
   END_RUNG wire#w15
   RUNG wire#powerrail
      Contact( #statUnitStatus.state.execute )
      Contact( #unitStatus.specialFunctions.GaugeRnR1CathodeStack )
      Contact( #instGaugeRnR1StackMainPnPMoveReelCutConvyorAlignTableJob21.jobStatus.completed )
   END_RUNG wire#w16
   RUNG wire#powerrail
      #instGaugeRnR1StackMainPnPMoveAlignTableJob23(interlock := wire#w17, startCondition := wire#w18, parentReferenceDesignator := "Unit1.Em5.Config".em.referenceDesignator.combined, jobNumber := "U1EM5_JOB23", singleCycleJob := TRUE, hmiInterface := "Unit1.Em5.HmiInterface".gaugeRnR.jobs, jobs := "Unit1.Em5.ControlNodes".gaugeRnR.jobs, jobStatus =>)
   END_RUNG
   RUNG wire#powerrail
      Contact( "Unit1.Em5.ControlNodes".em.status.initialized )
   END_RUNG wire#w17
   RUNG wire#powerrail
      Contact( #statUnitStatus.state.execute )
      Contact( #unitStatus.specialFunctions.GaugeRnR1CathodeStack )
      Contact( #instGaugeRnR1StackMainPnP2ToAlignTableJob22.jobStatus.completed )
   END_RUNG wire#w18
   RUNG wire#powerrail
      #instGaugeRnR1StackAlignTableToMainPnP1Job24(interlock := wire#w19, startCondition := wire#w20, parentReferenceDesignator := "Unit1.Em5.Config".em.referenceDesignator.combined, jobNumber := "U1EM5_JOB24", singleCycleJob := TRUE, hmiInterface := "Unit1.Em5.HmiInterface".gaugeRnR.jobs, jobs := "Unit1.Em5.ControlNodes".gaugeRnR.jobs, jobStatus =>)
   END_RUNG
   RUNG wire#powerrail
      Contact( "Unit1.Em5.ControlNodes".em.status.initialized )
   END_RUNG wire#w19
   RUNG wire#powerrail
      Contact( #statUnitStatus.state.execute )
      Contact( #unitStatus.specialFunctions.GaugeRnR1CathodeStack )
      Contact( #instGaugeRnR1StackMainPnPMoveAlignTableJob23.jobStatus.completed )
   END_RUNG wire#w20
   RUNG wire#powerrail
      #instGaugeRnR1StackMainPnPMoveReelCutConvyorAlignTableJob25(interlock := wire#w21, startCondition := wire#w22, parentReferenceDesignator := "Unit1.Em5.Config".em.referenceDesignator.combined, jobNumber := "U1EM5_JOB25", singleCycleJob := TRUE, hmiInterface := "Unit1.Em5.HmiInterface".gaugeRnR.jobs, jobs := "Unit1.Em5.ControlNodes".gaugeRnR.jobs, jobStatus =>)
   END_RUNG
   RUNG wire#powerrail
      Contact( "Unit1.Em5.ControlNodes".em.status.initialized )
   END_RUNG wire#w21
   RUNG wire#powerrail
      Contact( #statUnitStatus.state.execute )
      Contact( #unitStatus.specialFunctions.GaugeRnR1CathodeStack )
      Contact( #instGaugeRnR1StackAlignTableToMainPnP1Job24.jobStatus.completed )
   END_RUNG wire#w22
   RUNG wire#powerrail
      #instGaugeRnR1StackUnloadMasterPieceJob26(interlock := wire#w23, startCondition := wire#w24, parentReferenceDesignator := "Unit1.Em5.Config".em.referenceDesignator.combined, jobNumber := "U1EM5_JOB26", singleCycleJob := TRUE, hmiInterface := "Unit1.Em5.HmiInterface".gaugeRnR.jobs, jobs := "Unit1.Em5.ControlNodes".gaugeRnR.jobs, jobStatus =>)
   END_RUNG
   RUNG wire#powerrail
      Contact( "Unit1.Em5.ControlNodes".em.status.initialized )
   END_RUNG wire#w23
   RUNG wire#powerrail
      Contact( #statUnitStatus.state.execute )
      Contact( #unitStatus.specialFunctions.GaugeRnR1CathodeStack )
      Contact( #instGaugeRnR1StackMainPnPMoveReelCutConvyorAlignTableJob25.jobStatus.completed )
   END_RUNG wire#w24
   // the same network as SCL:
   #instGaugeRnR1StackMainPnPMoveReelCutConvyorAlignTableJob15(parentReferenceDesignator := "Unit1.Em5.Config".em.referenceDesignator.combined,   // "LAF_SelectJob"
                           jobNumber := "U1EM5_JOB15",
                           singleCycleJob := TRUE,
                           interlock := "Unit1.Em5.ControlNodes".em.status.initialized,
                           startCondition := #statUnitStatus.state.execute AND #unitStatus.specialFunctions.GaugeRnR1CathodeStack AND #instGaugeRnRCommonAlignTableVisionAdjustJob6.jobStatus.completed,
                           hmiInterface := "Unit1.Em5.HmiInterface".gaugeRnR.jobs,
                           jobs := "Unit1.Em5.ControlNodes".gaugeRnR.jobs);
   #instGaugeRnR1StackAlignTableToMainPnP2Job16(parentReferenceDesignator := "Unit1.Em5.Config".em.referenceDesignator.combined,   // "LAF_SelectJob"
                           jobNumber := "U1EM5_JOB16",
                           singleCycleJob := TRUE,
                           interlock := "Unit1.Em5.ControlNodes".em.status.initialized,
                           startCondition := #statUnitStatus.state.execute AND #unitStatus.specialFunctions.GaugeRnR1CathodeStack AND #instGaugeRnR1StackMainPnPMoveReelCutConvyorAlignTableJob15.jobStatus.completed,
                           hmiInterface := "Unit1.Em5.HmiInterface".gaugeRnR.jobs,
                           jobs := "Unit1.Em5.ControlNodes".gaugeRnR.jobs);
   #instGaugeRnR1StackMainPnPMoveAlignTableJob17(parentReferenceDesignator := "Unit1.Em5.Config".em.referenceDesignator.combined,   // "LAF_SelectJob"
                           jobNumber := "U1EM5_JOB17",
                           singleCycleJob := TRUE,
                           interlock := "Unit1.Em5.ControlNodes".em.status.initialized,
                           startCondition := #statUnitStatus.state.execute AND #unitStatus.specialFunctions.GaugeRnR1CathodeStack AND #instGaugeRnR1StackAlignTableToMainPnP2Job16.jobStatus.completed,
                           hmiInterface := "Unit1.Em5.HmiInterface".gaugeRnR.jobs,
                           jobs := "Unit1.Em5.ControlNodes".gaugeRnR.jobs);
   #instGaugeRnR1StackAlignTableMoveWaitJob18(parentReferenceDesignator := "Unit1.Em5.Config".em.referenceDesignator.combined,   // "LAF_SelectJob"
                           jobNumber := "U1EM5_JOB18",
                           singleCycleJob := TRUE,
                           interlock := "Unit1.Em5.ControlNodes".em.status.initialized,
                           startCondition := #statUnitStatus.state.execute AND #unitStatus.specialFunctions.GaugeRnR1CathodeStack AND #instGaugeRnR1StackMainPnPMoveAlignTableJob17.jobStatus.completed,
                           hmiInterface := "Unit1.Em5.HmiInterface".gaugeRnR.jobs,
                           jobs := "Unit1.Em5.ControlNodes".gaugeRnR.jobs);
   #instGaugeRnR1StackMainPnP2ToStackTableJob19(parentReferenceDesignator := "Unit1.Em5.Config".em.referenceDesignator.combined,   // "LAF_SelectJob"
                           jobNumber := "U1EM5_JOB19",
                           singleCycleJob := TRUE,
                           interlock := "Unit1.Em5.ControlNodes".em.status.initialized,
                           startCondition := #statUnitStatus.state.execute AND #unitStatus.specialFunctions.GaugeRnR1CathodeStack AND #instGaugeRnR1StackAlignTableMoveWaitJob18.jobStatus.completed,
                           hmiInterface := "Unit1.Em5.HmiInterface".gaugeRnR.jobs,
                           jobs := "Unit1.Em5.ControlNodes".gaugeRnR.jobs);
   #instGaugeRnR1StackStackTableToMainPnP2Job20(parentReferenceDesignator := "Unit1.Em5.Config".em.referenceDesignator.combined,   // "LAF_SelectJob"
                           jobNumber := "U1EM5_JOB20",
                           singleCycleJob := TRUE,
                           interlock := "Unit1.Em5.ControlNodes".em.status.initialized,
                           startCondition := #statUnitStatus.state.execute AND #unitStatus.specialFunctions.GaugeRnR1CathodeStack AND #instGaugeRnR1StackMainPnP2ToStackTableJob19.jobStatus.completed AND "Unit1.EmNodes".emRelations.em06.sequence.Spare2.jobInterface[3].workingDone,
                           hmiInterface := "Unit1.Em5.HmiInterface".gaugeRnR.jobs,
                           jobs := "Unit1.Em5.ControlNodes".gaugeRnR.jobs);
   #instGaugeRnR1StackMainPnPMoveReelCutConvyorAlignTableJob21(parentReferenceDesignator := "Unit1.Em5.Config".em.referenceDesignator.combined,   // "LAF_SelectJob"
                           jobNumber := "U1EM5_JOB21",
                           singleCycleJob := TRUE,
                           interlock := "Unit1.Em5.ControlNodes".em.status.initialized,
                           startCondition := #statUnitStatus.state.execute AND #unitStatus.specialFunctions.GaugeRnR1CathodeStack AND #instGaugeRnR1StackStackTableToMainPnP2Job20.jobStatus.completed,
                           hmiInterface := "Unit1.Em5.HmiInterface".gaugeRnR.jobs,
                           jobs := "Unit1.Em5.ControlNodes".gaugeRnR.jobs);
   #instGaugeRnR1StackMainPnP2ToAlignTableJob22(parentReferenceDesignator := "Unit1.Em5.Config".em.referenceDesignator.combined,   // "LAF_SelectJob"
                           jobNumber := "U1EM5_JOB22",
                           singleCycleJob := TRUE,
                           interlock := "Unit1.Em5.ControlNodes".em.status.initialized,
                           startCondition := #statUnitStatus.state.execute AND #unitStatus.specialFunctions.GaugeRnR1CathodeStack AND #instGaugeRnR1StackMainPnPMoveReelCutConvyorAlignTableJob21.jobStatus.completed,
                           hmiInterface := "Unit1.Em5.HmiInterface".gaugeRnR.jobs,
                           jobs := "Unit1.Em5.ControlNodes".gaugeRnR.jobs);
   #instGaugeRnR1StackMainPnPMoveAlignTableJob23(parentReferenceDesignator := "Unit1.Em5.Config".em.referenceDesignator.combined,   // "LAF_SelectJob"
                           jobNumber := "U1EM5_JOB23",
                           singleCycleJob := TRUE,
                           interlock := "Unit1.Em5.ControlNodes".em.status.initialized,
                           startCondition := #statUnitStatus.state.execute AND #unitStatus.specialFunctions.GaugeRnR1CathodeStack AND #instGaugeRnR1StackMainPnP2ToAlignTableJob22.jobStatus.completed,
                           hmiInterface := "Unit1.Em5.HmiInterface".gaugeRnR.jobs,
                           jobs := "Unit1.Em5.ControlNodes".gaugeRnR.jobs);
   #instGaugeRnR1StackAlignTableToMainPnP1Job24(parentReferenceDesignator := "Unit1.Em5.Config".em.referenceDesignator.combined,   // "LAF_SelectJob"
                           jobNumber := "U1EM5_JOB24",
                           singleCycleJob := TRUE,
                           interlock := "Unit1.Em5.ControlNodes".em.status.initialized,
                           startCondition := #statUnitStatus.state.execute AND #unitStatus.specialFunctions.GaugeRnR1CathodeStack AND #instGaugeRnR1StackMainPnPMoveAlignTableJob23.jobStatus.completed,
                           hmiInterface := "Unit1.Em5.HmiInterface".gaugeRnR.jobs,
                           jobs := "Unit1.Em5.ControlNodes".gaugeRnR.jobs);
   #instGaugeRnR1StackMainPnPMoveReelCutConvyorAlignTableJob25(parentReferenceDesignator := "Unit1.Em5.Config".em.referenceDesignator.combined,   // "LAF_SelectJob"
                           jobNumber := "U1EM5_JOB25",
                           singleCycleJob := TRUE,
                           interlock := "Unit1.Em5.ControlNodes".em.status.initialized,
                           startCondition := #statUnitStatus.state.execute AND #unitStatus.specialFunctions.GaugeRnR1CathodeStack AND #instGaugeRnR1StackAlignTableToMainPnP1Job24.jobStatus.completed,
                           hmiInterface := "Unit1.Em5.HmiInterface".gaugeRnR.jobs,
                           jobs := "Unit1.Em5.ControlNodes".gaugeRnR.jobs);
   #instGaugeRnR1StackUnloadMasterPieceJob26(parentReferenceDesignator := "Unit1.Em5.Config".em.referenceDesignator.combined,   // "LAF_SelectJob"
                           jobNumber := "U1EM5_JOB26",
                           singleCycleJob := TRUE,
                           interlock := "Unit1.Em5.ControlNodes".em.status.initialized,
                           startCondition := #statUnitStatus.state.execute AND #unitStatus.specialFunctions.GaugeRnR1CathodeStack AND #instGaugeRnR1StackMainPnPMoveReelCutConvyorAlignTableJob25.jobStatus.completed,
                           hmiInterface := "Unit1.Em5.HmiInterface".gaugeRnR.jobs,
                           jobs := "Unit1.Em5.ControlNodes".gaugeRnR.jobs);
END_REGION

REGION Network 58: Gauge RnR 3 Stack Select Job
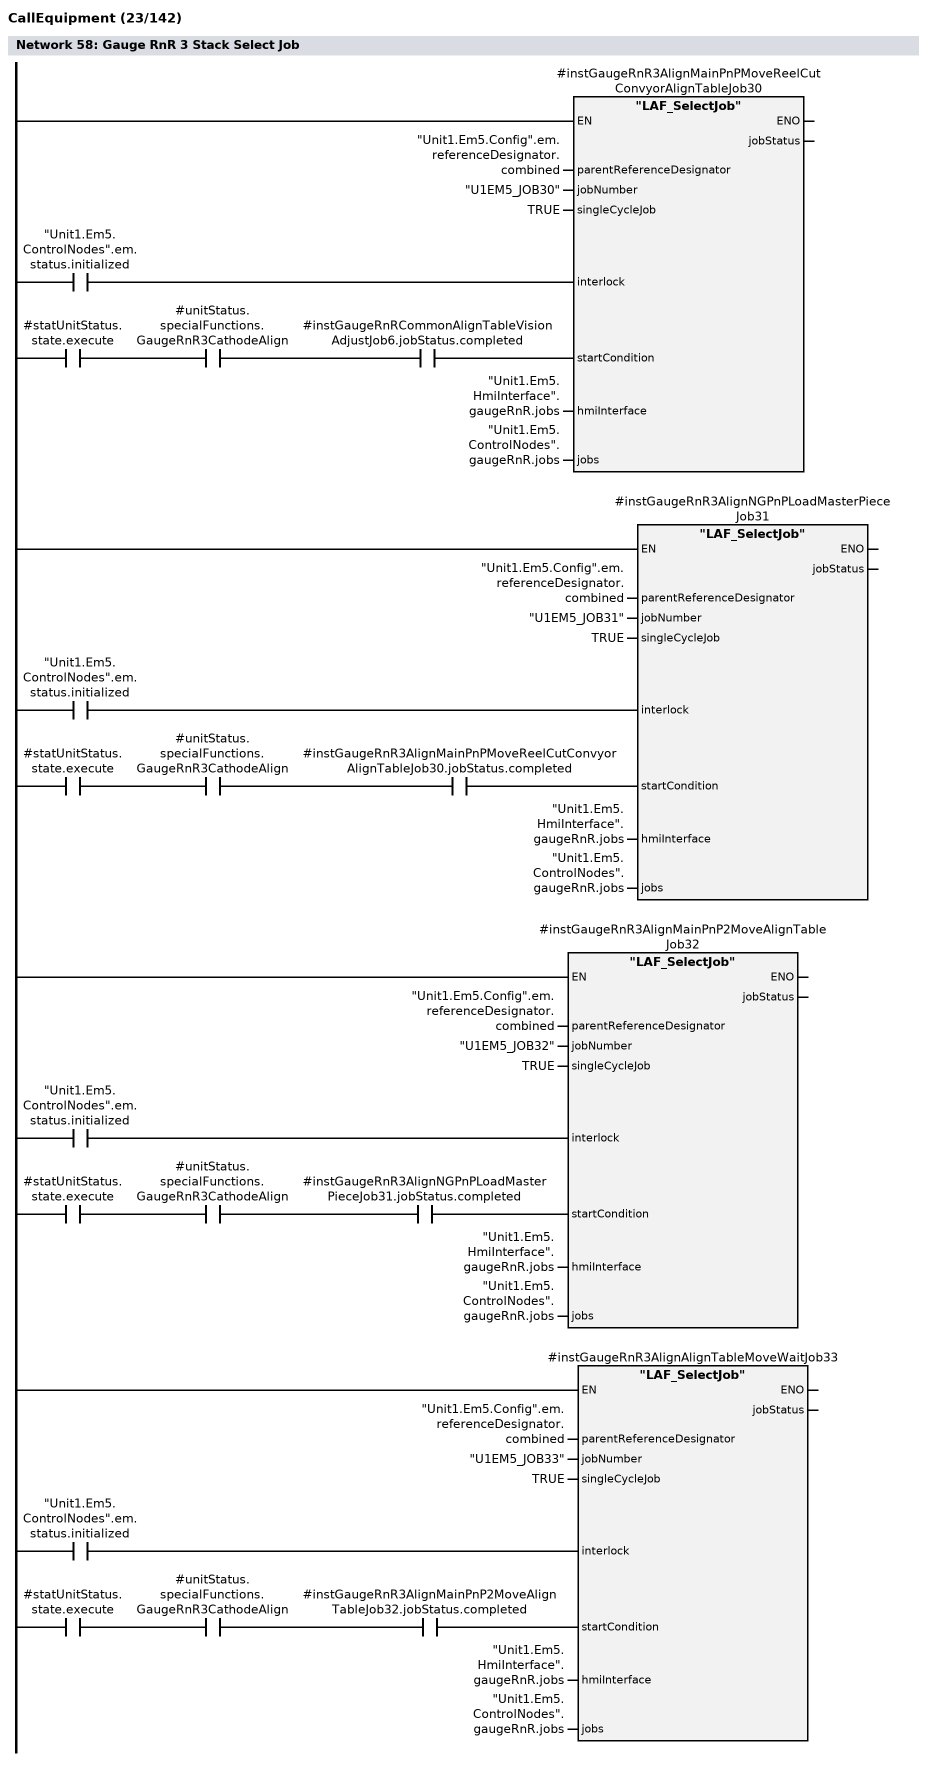
   RUNG wire#powerrail
      #instGaugeRnR3AlignMainPnPMoveReelCutConvyorAlignTableJob30(interlock := wire#w1, startCondition := wire#w2, parentReferenceDesignator := "Unit1.Em5.Config".em.referenceDesignator.combined, jobNumber := "U1EM5_JOB30", singleCycleJob := TRUE, hmiInterface := "Unit1.Em5.HmiInterface".gaugeRnR.jobs, jobs := "Unit1.Em5.ControlNodes".gaugeRnR.jobs, jobStatus =>)
   END_RUNG
   RUNG wire#powerrail
      Contact( "Unit1.Em5.ControlNodes".em.status.initialized )
   END_RUNG wire#w1
   RUNG wire#powerrail
      Contact( #statUnitStatus.state.execute )
      Contact( #unitStatus.specialFunctions.GaugeRnR3CathodeAlign )
      Contact( #instGaugeRnRCommonAlignTableVisionAdjustJob6.jobStatus.completed )
   END_RUNG wire#w2
   RUNG wire#powerrail
      #instGaugeRnR3AlignNGPnPLoadMasterPieceJob31(interlock := wire#w3, startCondition := wire#w4, parentReferenceDesignator := "Unit1.Em5.Config".em.referenceDesignator.combined, jobNumber := "U1EM5_JOB31", singleCycleJob := TRUE, hmiInterface := "Unit1.Em5.HmiInterface".gaugeRnR.jobs, jobs := "Unit1.Em5.ControlNodes".gaugeRnR.jobs, jobStatus =>)
   END_RUNG
   RUNG wire#powerrail
      Contact( "Unit1.Em5.ControlNodes".em.status.initialized )
   END_RUNG wire#w3
   RUNG wire#powerrail
      Contact( #statUnitStatus.state.execute )
      Contact( #unitStatus.specialFunctions.GaugeRnR3CathodeAlign )
      Contact( #instGaugeRnR3AlignMainPnPMoveReelCutConvyorAlignTableJob30.jobStatus.completed )
   END_RUNG wire#w4
   RUNG wire#powerrail
      #instGaugeRnR3AlignMainPnP2MoveAlignTableJob32(interlock := wire#w5, startCondition := wire#w6, parentReferenceDesignator := "Unit1.Em5.Config".em.referenceDesignator.combined, jobNumber := "U1EM5_JOB32", singleCycleJob := TRUE, hmiInterface := "Unit1.Em5.HmiInterface".gaugeRnR.jobs, jobs := "Unit1.Em5.ControlNodes".gaugeRnR.jobs, jobStatus =>)
   END_RUNG
   RUNG wire#powerrail
      Contact( "Unit1.Em5.ControlNodes".em.status.initialized )
   END_RUNG wire#w5
   RUNG wire#powerrail
      Contact( #statUnitStatus.state.execute )
      Contact( #unitStatus.specialFunctions.GaugeRnR3CathodeAlign )
      Contact( #instGaugeRnR3AlignNGPnPLoadMasterPieceJob31.jobStatus.completed )
   END_RUNG wire#w6
   RUNG wire#powerrail
      #instGaugeRnR3AlignAlignTableMoveWaitJob33(interlock := wire#w7, startCondition := wire#w8, parentReferenceDesignator := "Unit1.Em5.Config".em.referenceDesignator.combined, jobNumber := "U1EM5_JOB33", singleCycleJob := TRUE, hmiInterface := "Unit1.Em5.HmiInterface".gaugeRnR.jobs, jobs := "Unit1.Em5.ControlNodes".gaugeRnR.jobs, jobStatus =>)
   END_RUNG
   RUNG wire#powerrail
      Contact( "Unit1.Em5.ControlNodes".em.status.initialized )
   END_RUNG wire#w7
   RUNG wire#powerrail
      Contact( #statUnitStatus.state.execute )
      Contact( #unitStatus.specialFunctions.GaugeRnR3CathodeAlign )
      Contact( #instGaugeRnR3AlignMainPnP2MoveAlignTableJob32.jobStatus.completed )
   END_RUNG wire#w8
   // the same network as SCL:
   #instGaugeRnR3AlignMainPnPMoveReelCutConvyorAlignTableJob30(parentReferenceDesignator := "Unit1.Em5.Config".em.referenceDesignator.combined,   // "LAF_SelectJob"
                           jobNumber := "U1EM5_JOB30",
                           singleCycleJob := TRUE,
                           interlock := "Unit1.Em5.ControlNodes".em.status.initialized,
                           startCondition := #statUnitStatus.state.execute AND #unitStatus.specialFunctions.GaugeRnR3CathodeAlign AND #instGaugeRnRCommonAlignTableVisionAdjustJob6.jobStatus.completed,
                           hmiInterface := "Unit1.Em5.HmiInterface".gaugeRnR.jobs,
                           jobs := "Unit1.Em5.ControlNodes".gaugeRnR.jobs);
   #instGaugeRnR3AlignNGPnPLoadMasterPieceJob31(parentReferenceDesignator := "Unit1.Em5.Config".em.referenceDesignator.combined,   // "LAF_SelectJob"
                           jobNumber := "U1EM5_JOB31",
                           singleCycleJob := TRUE,
                           interlock := "Unit1.Em5.ControlNodes".em.status.initialized,
                           startCondition := #statUnitStatus.state.execute AND #unitStatus.specialFunctions.GaugeRnR3CathodeAlign AND #instGaugeRnR3AlignMainPnPMoveReelCutConvyorAlignTableJob30.jobStatus.completed,
                           hmiInterface := "Unit1.Em5.HmiInterface".gaugeRnR.jobs,
                           jobs := "Unit1.Em5.ControlNodes".gaugeRnR.jobs);
   #instGaugeRnR3AlignMainPnP2MoveAlignTableJob32(parentReferenceDesignator := "Unit1.Em5.Config".em.referenceDesignator.combined,   // "LAF_SelectJob"
                           jobNumber := "U1EM5_JOB32",
                           singleCycleJob := TRUE,
                           interlock := "Unit1.Em5.ControlNodes".em.status.initialized,
                           startCondition := #statUnitStatus.state.execute AND #unitStatus.specialFunctions.GaugeRnR3CathodeAlign AND #instGaugeRnR3AlignNGPnPLoadMasterPieceJob31.jobStatus.completed,
                           hmiInterface := "Unit1.Em5.HmiInterface".gaugeRnR.jobs,
                           jobs := "Unit1.Em5.ControlNodes".gaugeRnR.jobs);
   #instGaugeRnR3AlignAlignTableMoveWaitJob33(parentReferenceDesignator := "Unit1.Em5.Config".em.referenceDesignator.combined,   // "LAF_SelectJob"
                           jobNumber := "U1EM5_JOB33",
                           singleCycleJob := TRUE,
                           interlock := "Unit1.Em5.ControlNodes".em.status.initialized,
                           startCondition := #statUnitStatus.state.execute AND #unitStatus.specialFunctions.GaugeRnR3CathodeAlign AND #instGaugeRnR3AlignMainPnP2MoveAlignTableJob32.jobStatus.completed,
                           hmiInterface := "Unit1.Em5.HmiInterface".gaugeRnR.jobs,
                           jobs := "Unit1.Em5.ControlNodes".gaugeRnR.jobs);
END_REGION

REGION Network 59: Gauge RnR Job 1 Interface
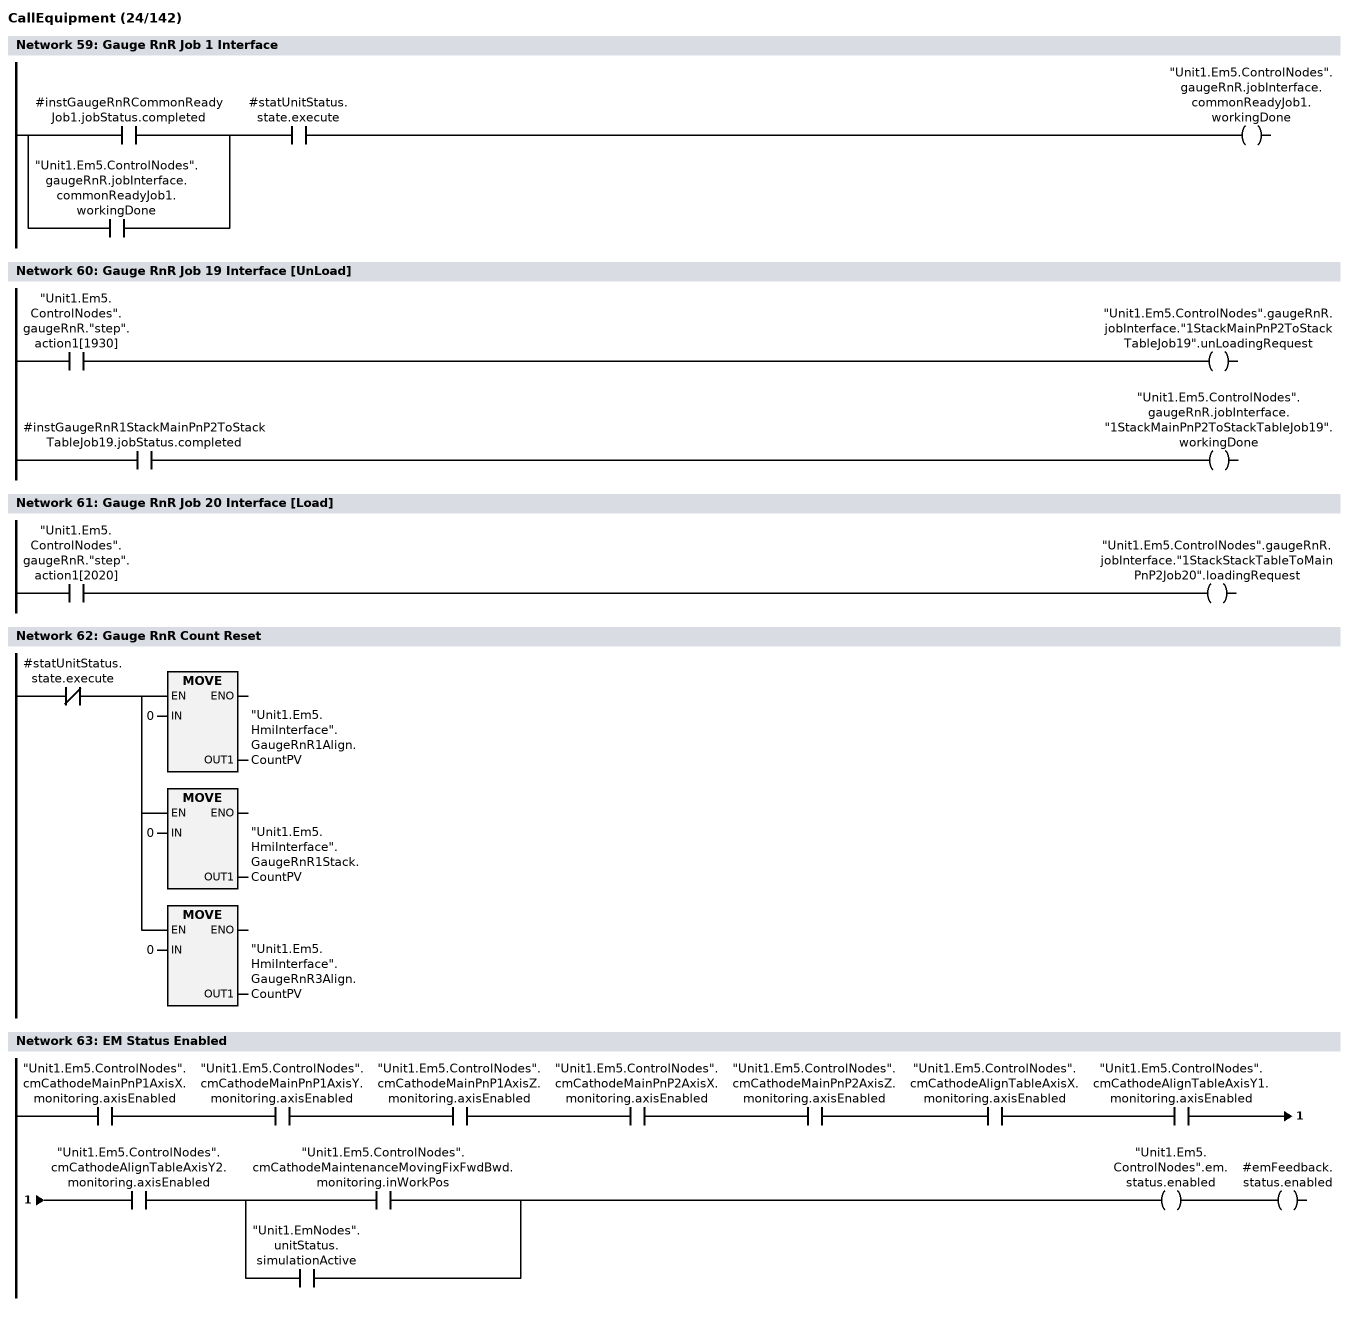
   RUNG wire#powerrail
      Contact( #instGaugeRnRCommonReadyJob1.jobStatus.completed )
      wire#w1
      Contact( #statUnitStatus.state.execute )
      Coil( "Unit1.Em5.ControlNodes".gaugeRnR.jobInterface.commonReadyJob1.workingDone )
   END_RUNG
   RUNG wire#powerrail
      Contact( "Unit1.Em5.ControlNodes".gaugeRnR.jobInterface.commonReadyJob1.workingDone )
   END_RUNG wire#w1
   // the same network as SCL:
   "Unit1.Em5.ControlNodes".gaugeRnR.jobInterface.commonReadyJob1.workingDone := (#instGaugeRnRCommonReadyJob1.jobStatus.completed OR "Unit1.Em5.ControlNodes".gaugeRnR.jobInterface.commonReadyJob1.workingDone) AND #statUnitStatus.state.execute;
END_REGION

REGION Network 60: Gauge RnR Job 19 Interface [UnLoad]
   RUNG wire#powerrail
      Contact( "Unit1.Em5.ControlNodes".gaugeRnR."step".action1[1930] )
      Coil( "Unit1.Em5.ControlNodes".gaugeRnR.jobInterface."1StackMainPnP2ToStackTableJob19".unLoadingRequest )
   END_RUNG
   RUNG wire#powerrail
      Contact( #instGaugeRnR1StackMainPnP2ToStackTableJob19.jobStatus.completed )
      Coil( "Unit1.Em5.ControlNodes".gaugeRnR.jobInterface."1StackMainPnP2ToStackTableJob19".workingDone )
   END_RUNG
   // the same network as SCL:
   "Unit1.Em5.ControlNodes".gaugeRnR.jobInterface."1StackMainPnP2ToStackTableJob19".unLoadingRequest := "Unit1.Em5.ControlNodes".gaugeRnR."step".action1[1930];
   "Unit1.Em5.ControlNodes".gaugeRnR.jobInterface."1StackMainPnP2ToStackTableJob19".workingDone := #instGaugeRnR1StackMainPnP2ToStackTableJob19.jobStatus.completed;
END_REGION

REGION Network 61: Gauge RnR Job 20 Interface [Load]
   RUNG wire#powerrail
      Contact( "Unit1.Em5.ControlNodes".gaugeRnR."step".action1[2020] )
      Coil( "Unit1.Em5.ControlNodes".gaugeRnR.jobInterface."1StackStackTableToMainPnP2Job20".loadingRequest )
   END_RUNG
   // the same network as SCL:
   "Unit1.Em5.ControlNodes".gaugeRnR.jobInterface."1StackStackTableToMainPnP2Job20".loadingRequest := "Unit1.Em5.ControlNodes".gaugeRnR."step".action1[2020];
END_REGION

REGION Network 62: Gauge RnR Count Reset
   RUNG wire#powerrail
      I_Contact( #statUnitStatus.state.execute )
      wire#w1
      Move(in := 0, out1 => "Unit1.Em5.HmiInterface".GaugeRnR1Align.CountPV)
   END_RUNG
   RUNG wire#w1
      Move(in := 0, out1 => "Unit1.Em5.HmiInterface".GaugeRnR1Stack.CountPV)
   END_RUNG
   RUNG wire#w1
      Move(in := 0, out1 => "Unit1.Em5.HmiInterface".GaugeRnR3Align.CountPV)
   END_RUNG
   // the same network as SCL:
   IF NOT #statUnitStatus.state.execute THEN
       "Unit1.Em5.HmiInterface".GaugeRnR1Align.CountPV := 0;
       "Unit1.Em5.HmiInterface".GaugeRnR1Stack.CountPV := 0;
       "Unit1.Em5.HmiInterface".GaugeRnR3Align.CountPV := 0;
   END_IF;
END_REGION

REGION Network 63: EM Status Enabled
   RUNG wire#powerrail
      Contact( "Unit1.Em5.ControlNodes".cmCathodeMainPnP1AxisX.monitoring.axisEnabled )
      Contact( "Unit1.Em5.ControlNodes".cmCathodeMainPnP1AxisY.monitoring.axisEnabled )
      Contact( "Unit1.Em5.ControlNodes".cmCathodeMainPnP1AxisZ.monitoring.axisEnabled )
      Contact( "Unit1.Em5.ControlNodes".cmCathodeMainPnP2AxisX.monitoring.axisEnabled )
      Contact( "Unit1.Em5.ControlNodes".cmCathodeMainPnP2AxisZ.monitoring.axisEnabled )
      Contact( "Unit1.Em5.ControlNodes".cmCathodeAlignTableAxisX.monitoring.axisEnabled )
      Contact( "Unit1.Em5.ControlNodes".cmCathodeAlignTableAxisY1.monitoring.axisEnabled )
      Contact( "Unit1.Em5.ControlNodes".cmCathodeAlignTableAxisY2.monitoring.axisEnabled )
      wire#w1
      Contact( "Unit1.Em5.ControlNodes".cmCathodeMaintenanceMovingFixFwdBwd.monitoring.inWorkPos )
      wire#w2
      Coil( "Unit1.Em5.ControlNodes".em.status.enabled )
      Coil( #emFeedback.status.enabled )
   END_RUNG
   RUNG wire#w1
      Contact( "Unit1.EmNodes".unitStatus.simulationActive )
   END_RUNG wire#w2
   // the same network as SCL:
   "Unit1.Em5.ControlNodes".em.status.enabled := "Unit1.Em5.ControlNodes".cmCathodeMainPnP1AxisX.monitoring.axisEnabled AND "Unit1.Em5.ControlNodes".cmCathodeMainPnP1AxisY.monitoring.axisEnabled AND "Unit1.Em5.ControlNodes".cmCathodeMainPnP1AxisZ.monitoring.axisEnabled AND "Unit1.Em5.ControlNodes".cmCathodeMainPnP2AxisX.monitoring.axisEnabled AND "Unit1.Em5.ControlNodes".cmCathodeMainPnP2AxisZ.monitoring.axisEnabled AND "Unit1.Em5.ControlNodes".cmCathodeAlignTableAxisX.monitoring.axisEnabled AND "Unit1.Em5.ControlNodes".cmCathodeAlignTableAxisY1.monitoring.axisEnabled AND "Unit1.Em5.ControlNodes".cmCathodeAlignTableAxisY2.monitoring.axisEnabled AND ("Unit1.Em5.ControlNodes".cmCathodeMaintenanceMovingFixFwdBwd.monitoring.inWorkPos OR "Unit1.EmNodes".unitStatus.simulationActive);
   #emFeedback.status.enabled := "Unit1.Em5.ControlNodes".em.status.enabled;
END_REGION

REGION Network 64: Set EM To Initialized
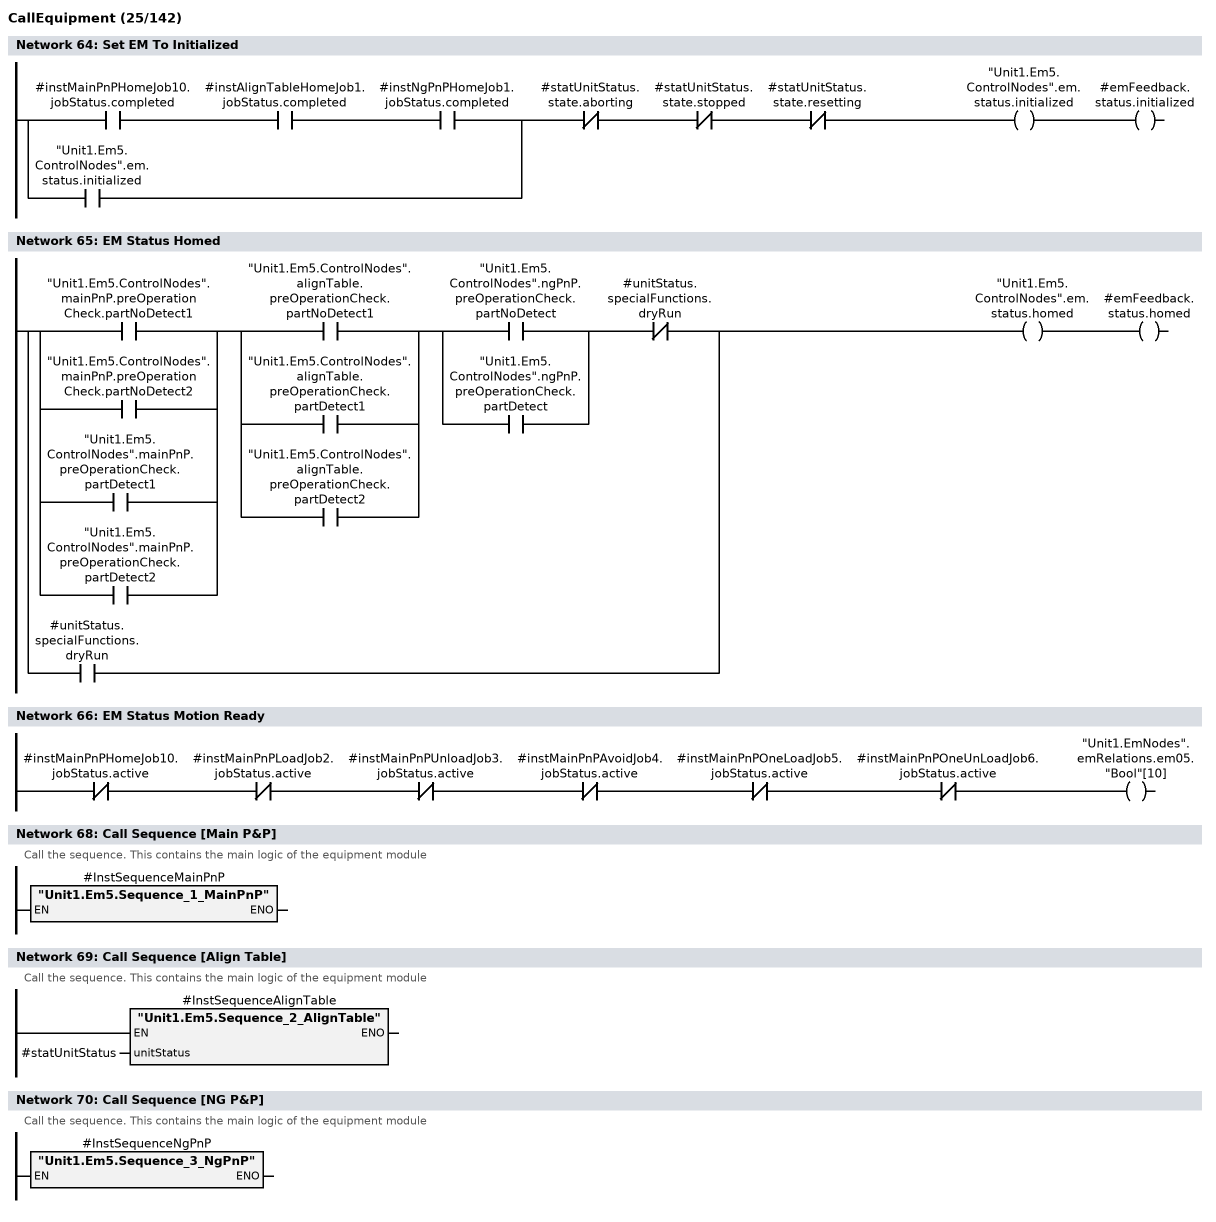
   RUNG wire#powerrail
      Contact( #instMainPnPHomeJob10.jobStatus.completed )
      Contact( #instAlignTableHomeJob1.jobStatus.completed )
      Contact( #instNgPnPHomeJob1.jobStatus.completed )
      wire#w1
      I_Contact( #statUnitStatus.state.aborting )
      I_Contact( #statUnitStatus.state.stopped )
      I_Contact( #statUnitStatus.state.resetting )
      Coil( "Unit1.Em5.ControlNodes".em.status.initialized )
      Coil( #emFeedback.status.initialized )
   END_RUNG
   RUNG wire#powerrail
      Contact( "Unit1.Em5.ControlNodes".em.status.initialized )
   END_RUNG wire#w1
   // the same network as SCL:
   "Unit1.Em5.ControlNodes".em.status.initialized := ((#instMainPnPHomeJob10.jobStatus.completed AND #instAlignTableHomeJob1.jobStatus.completed AND #instNgPnPHomeJob1.jobStatus.completed) OR "Unit1.Em5.ControlNodes".em.status.initialized) AND NOT #statUnitStatus.state.aborting AND NOT #statUnitStatus.state.stopped AND NOT #statUnitStatus.state.resetting;
   #emFeedback.status.initialized := "Unit1.Em5.ControlNodes".em.status.initialized;
END_REGION

REGION Network 65: EM Status Homed
   RUNG wire#powerrail
      Contact( "Unit1.Em5.ControlNodes".mainPnP.preOperationCheck.partNoDetect1 )
      wire#w1
      Contact( "Unit1.Em5.ControlNodes".alignTable.preOperationCheck.partNoDetect1 )
      wire#w2
      Contact( "Unit1.Em5.ControlNodes".ngPnP.preOperationCheck.partNoDetect )
      wire#w3
      I_Contact( #unitStatus.specialFunctions.dryRun )
      wire#w4
      Coil( "Unit1.Em5.ControlNodes".em.status.homed )
      Coil( #emFeedback.status.homed )
   END_RUNG
   RUNG wire#powerrail
      Contact( "Unit1.Em5.ControlNodes".mainPnP.preOperationCheck.partNoDetect2 )
   END_RUNG wire#w1
   RUNG wire#powerrail
      Contact( "Unit1.Em5.ControlNodes".mainPnP.preOperationCheck.partDetect1 )
   END_RUNG wire#w1
   RUNG wire#powerrail
      Contact( "Unit1.Em5.ControlNodes".mainPnP.preOperationCheck.partDetect2 )
   END_RUNG wire#w1
   RUNG wire#w1
      Contact( "Unit1.Em5.ControlNodes".alignTable.preOperationCheck.partDetect1 )
   END_RUNG wire#w2
   RUNG wire#w1
      Contact( "Unit1.Em5.ControlNodes".alignTable.preOperationCheck.partDetect2 )
   END_RUNG wire#w2
   RUNG wire#w2
      Contact( "Unit1.Em5.ControlNodes".ngPnP.preOperationCheck.partDetect )
   END_RUNG wire#w3
   RUNG wire#powerrail
      Contact( #unitStatus.specialFunctions.dryRun )
   END_RUNG wire#w4
   // the same network as SCL:
   "Unit1.Em5.ControlNodes".em.status.homed := (("Unit1.Em5.ControlNodes".mainPnP.preOperationCheck.partNoDetect1 OR "Unit1.Em5.ControlNodes".mainPnP.preOperationCheck.partNoDetect2 OR "Unit1.Em5.ControlNodes".mainPnP.preOperationCheck.partDetect1 OR "Unit1.Em5.ControlNodes".mainPnP.preOperationCheck.partDetect2) AND ("Unit1.Em5.ControlNodes".alignTable.preOperationCheck.partNoDetect1 OR "Unit1.Em5.ControlNodes".alignTable.preOperationCheck.partDetect1 OR "Unit1.Em5.ControlNodes".alignTable.preOperationCheck.partDetect2) AND ("Unit1.Em5.ControlNodes".ngPnP.preOperationCheck.partNoDetect OR "Unit1.Em5.ControlNodes".ngPnP.preOperationCheck.partDetect) AND NOT #unitStatus.specialFunctions.dryRun) OR #unitStatus.specialFunctions.dryRun;
   #emFeedback.status.homed := "Unit1.Em5.ControlNodes".em.status.homed;
END_REGION

REGION Network 66: EM Status Motion Ready
   RUNG wire#powerrail
      I_Contact( #instMainPnPHomeJob10.jobStatus.active )
      I_Contact( #instMainPnPLoadJob2.jobStatus.active )
      I_Contact( #instMainPnPUnloadJob3.jobStatus.active )
      I_Contact( #instMainPnPAvoidJob4.jobStatus.active )
      I_Contact( #instMainPnPOneLoadJob5.jobStatus.active )
      I_Contact( #instMainPnPOneUnLoadJob6.jobStatus.active )
      Coil( "Unit1.EmNodes".emRelations.em05."Bool"[10] )
   END_RUNG
   // the same network as SCL:
   "Unit1.EmNodes".emRelations.em05."Bool"[10] := NOT #instMainPnPHomeJob10.jobStatus.active AND NOT #instMainPnPLoadJob2.jobStatus.active AND NOT #instMainPnPUnloadJob3.jobStatus.active AND NOT #instMainPnPAvoidJob4.jobStatus.active AND NOT #instMainPnPOneLoadJob5.jobStatus.active AND NOT #instMainPnPOneUnLoadJob6.jobStatus.active;
END_REGION

REGION Network 68: Call Sequence [Main P&P]
   // Call the sequence. This contains the main logic of the equipment module
   RUNG wire#powerrail
      #InstSequenceMainPnP()
   END_RUNG
   // the same network as SCL:
   #InstSequenceMainPnP();   // "Unit1.Em5.Sequence_1_MainPnP"
END_REGION

REGION Network 69: Call Sequence [Align Table]
   // Call the sequence. This contains the main logic of the equipment module
   RUNG wire#powerrail
      #InstSequenceAlignTable(unitStatus := #statUnitStatus)
   END_RUNG
   // the same network as SCL:
   #InstSequenceAlignTable(unitStatus := #statUnitStatus);   // "Unit1.Em5.Sequence_2_AlignTable"
END_REGION

REGION Network 70: Call Sequence [NG P&P]
   // Call the sequence. This contains the main logic of the equipment module
   RUNG wire#powerrail
      #InstSequenceNgPnP()
   END_RUNG
   // the same network as SCL:
   #InstSequenceNgPnP();   // "Unit1.Em5.Sequence_3_NgPnP"
END_REGION

REGION Network 71: Call Sequence [GuageRnR]
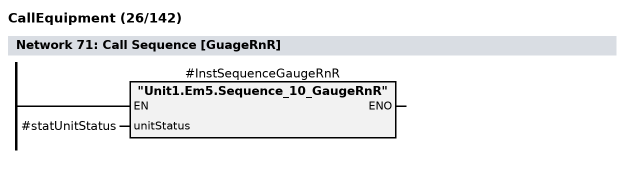
   RUNG wire#powerrail
      #InstSequenceGaugeRnR(unitStatus := #statUnitStatus)
   END_RUNG
   // the same network as SCL:
   #InstSequenceGaugeRnR(unitStatus := #statUnitStatus);   // "Unit1.Em5.Sequence_10_GaugeRnR"
END_REGION

REGION Network 72: *************** Control Modules (Axis) *******************
   // Call control modules that are actuators after the em logic (jobs and sequence), so that the latest commands are applied to the actuators.
END_REGION

